	12:	 IF    bIWrappingChannelPiston2_Home AND    bIWrappingChannelPiston3_Home   THEN
		bASet4Comp:=TRUE;
		bASet3Comp:=FALSE;
		bAWrappingCone23FwdCom1:=FALSE;
		b8thConesPushed:=TRUE;
		bAFilm1Loaded_24_8Cone:=FALSE;
		bAFilm1Loaded_24_7Cone:=FALSE;
		bASensorMonitorBit3:=FALSE;
		bAConeMissErrorAtWrpConvTemp5_24:=FALSE;
		TON_8_24(IN:=FALSE);
		bWrapConvStopped4_24:=FALSE;
		TON_9_24(in:=FALSE);
		bAWrapConeCyl23_24:=FALSE;
		step4:=0;
		END_IF   sMessage_Wrapping:='Check Wrapping Piston Home  2 & 3 Reed Switch';
END_CASE


IF bAFlimNotLoaded3 AND b2_4SetHmiSelected AND bErrorReset AND bAutoModeOn THEN step4:=10; bAFlimNotLoaded3:=FALSE;HmiFilmLoadErr:=''; END_IF






IF bA6conesPushed AND CounterTilt23.CV<=3 THEN
bANextLayerStarted:=TRUE;
END_IF


IF bA3Pushed OR bA6conesPushed AND bAFirstConeAtWrapConv THEN
bAConvStartInterlock:=TRUE;
ELSE
bAConvStartInterlock:=FALSE;
END_IF

(*

IF bAConvFirstStartUnitB THEN
baConveyerStarted:=TRUE;
END_IF
IF baConveyerStarted AND



*)




IF bIWrappingCone1 AND   InterLockCounter.CV = 0  AND NOT  bQWrappingConveyorMotor THEN
 Interlockfor_1Cone_24:=TRUE;
 ELSE
 Interlockfor_1Cone_24:=FALSE; END_IF


IF bIWrappingCone1 AND   InterLockCounter.CV = 4  AND NOT  bQWrappingConveyorMotor THEN
 Interlockfor_5Cone_24:=TRUE;
 ELSE
 Interlockfor_5Cone_24:=FALSE; END_IF

IF bIWrappingCone1 AND   InterLockCounter.CV = 6  AND NOT  bQWrappingConveyorMotor THEN
 Interlockfor_7Cone_24:=TRUE;
 ELSE
 Interlockfor_7Cone_24:=FALSE; END_IF

WrappingCone1RT(CLK:=( bIWrappingCone1 AND NOT Interlockfor_1Cone_24 AND NOT Interlockfor_5Cone_24 AND NOT Interlockfor_7Cone_24 ), Q=> );

WrappingConvRT(CLK:= bQWrappingConveyorMotor , Q=> );

IF  WrappingConvRT.Q THEN
bAWrapConvStarted:=TRUE;

END_IF

IF WrappingCone1RT.Q THEN WCS1Sensed:=TRUE; END_IF

IF WCS1Sensed  (* AND bAWrapConvStarted OR bConvRunning*)  THEN
bAInterlockCountStart:=TRUE;
ELSE
bAInterlockCountStart:=FALSE;
 END_IF


IF  bQWrappingConveyorMotor AND NOT bIWrappingCone1 AND bAutoModeOn THEN
WCS1Sensed:=FALSE;
END_IF

(*TON_6(IN:=WCS1Sensed , PT:=T#0.2s , Q=> , ET=> );

IF TON_6.Q THEN bAWrapConvStarted:=FALSE; (*TON_6(in:=FALSE);*)END_IF


IF InterLockCounter.CV = 2 AND bManualModeOn THEN
TimerStartBit:=TRUE;
bAWrapConvStarted:=FALSE;
TON_10(IN:=TimerStartBit , PT:=t#0.2s , Q=> , ET=> );

 END_IF


IF TON_10.Q AND bQWrappingConveyorMotor THEN
bConvRunning:=TRUE;(*TON_10(in:=FALSE);*)
END_IF*)




IF bRowStopperIntOver THEN
bSaelUnitIntOverTemp:=TRUE;
END_IF



                                                                   (*=============== Interlock Logic for  2*4 WCS conveyor===================*)


CASE step7 OF


	0:	IF bSaelUnitIntOverTemp AND b2_4SetHmiSelected  THEN                                    (*========= need to check for reset Logic=    step7:=0    =======*)
		Step7:=Step7+1;
		END_IF

	1:	bWCSStart1_24:=TRUE;
		Step7:=Step7+1;

	2:	IF  bASealConvEnd1_24 THEN
		bSaelUnitIntOverTemp:=FALSE;
		Step7:=Step7+1;
		END_IF

	3:	bWCSStart2_24:=TRUE;
		bASealConvEnd1_24:=FALSE;
		Step7:=Step7+1;


	4:	IF bASealConvEnd2_24  THEN
		Step7:=Step7+1;
		END_IF

	5:	bWCSStart3_24:=TRUE;
		bASealConvEnd2_24:=FALSE;
		Step7:=2;

END_CASE



IF NOT bIEmergencySwitch OR bStopHmi  OR bServoOff OR bIMcStop THEN

bAWrappingConvStartAuto3_23:=FALSE;
bAWrappingConvStartAuto4_23:=FALSE;
bAWrappingConvStartAuto3:=FALSE;
bAWrappingConvStartAuto4:=FALSE;
bAWrappingConvStartAuto5:=FALSE;


		bAWrappingCone123FwdCom:=FALSE;


SealingOver1:=FALSE;

bAFilm1Loaded:=FALSE;
bAFilm2Loaded:=FALSE;
bAFilm3Loaded:=FALSE;
		WrapConvStartDly(in:=FALSE);
		bAConvRunning1:=FALSE;
		bWrapConvStopped2:=FALSE;
		TON_3(IN:=FALSE);
		TON_13_24(in:=FALSE);
		TON_4_24(IN:=FALSE);
		TON_12_24(in:=FALSE);
		bAConeMissErrorAtWrpConvTemp1_24:=FALSE;
		bAConeMissErrorAtWrpConvTemp2_24:=FALSE;
		bAWrapConeCyl123:=FALSE;

bWrapConvStopped2:=FALSE;
bWrapConvStopped3_24:=FALSE;
bWrapConvStopped4_24:=FALSE;
bWrapConvStopped4_24exp:=FALSE;


bAWrappingConvStart1_23:=FALSE;
bAWrappingConvStart4_23:=FALSE;
bAWrappingConvStart1:=FALSE;
bAWrappingConvStart2:=FALSE;
bAWrappingConvStart3:=FALSE;
bAWrappingConvStart4:=FALSE;
bAWrappingConvStart5:=FALSE;

bAconvReayTemp:=FALSE;
bAconvReayTemp2:=FALSE;
bAconvReadyTemp3:=FALSE;
bAconvReadyTemp4:=FALSE;
bAconvReadyTemp5:=FALSE;

bAWrappingConvStart1_23:=FALSE;
bACheckWrappConvError1:=FALSE;
bACheckWrappConvError2:=FALSE;
bACheckWrappConvError3:=FALSE;
bACheckWrappConvError4:=FALSE;
bACheckWrappConvError5:=FALSE;

bAWrappingConvStartAuto:=FALSE;
bAWrappingConvStartAuto2:=FALSE;
 bAWrappingConvStartAuto3:=FALSE;

bQAWrappingConveyorMotor1:=FALSE;
 bQAWrappingConveyorMotor2:=FALSE;
bQAWrappingConveyorMotor3:=FALSE;
 bQAWrappingConveyorMotor4:=FALSE;
bQAWrappingConveyorMotor5:=FALSE;

WrapConvStartDly3_23(IN:= FALSE);

bAConvRunning1:=FALSE;
 bAConvStartBit:=FALSE;

bASensorMonitorBit1:=FALSE;
bASensorMonitorBit2:=FALSE;
 bASensorMonitorBit3:=FALSE;

bASet1Comp:=FALSE;
bASet3Comp:=FALSE;
bASet2Comp:=FALSE;
bASet4Comp:=FALSE;

bAWrapConeCyl3:=FALSE;
bAWrapConeCyl123:=FALSE;
bAWrapConeCyl23_24_1:=FALSE;
bAWrapConeCyl23_24:=FALSE;

WCS1Sensed:=FALSE;
bSaelUnitIntOver:=FALSE;


bASealConvEnd1:=FALSE;
bASealConvEnd2:=FALSE;

InterLockCounter.RESET:=TRUE;
bAWrappingCone123OnAuto:=FALSE;
bAWrappingCone123_23OnAuto:=FALSE;
bQAWrappingConveyorMotor4_23:=FALSE;
bQAWrappingConveyorMotor3_23:=FALSE;


bCount_ConvLockBit2:=FALSE;
bCount_ConvLockBit:=FALSE;
bASealConvEnd1_24:=FALSE;
bASealConvEnd2_24:=FALSE;
step1:=0;
step2:=0;
step3:=0;
step4:=0;
step5:=0;
step6:=0;
step7:=0;
bAConvStartBit:=FALSE;

bA3Pushed:=FALSE;
b4thConePushed:=FALSE;
b6thConePushed_24:=FALSE;

bWCSStart1_24:=FALSE;
bWCSStart2_24:=FALSE;
bWCSStart3_24:=FALSE;

TON_6_24(IN:=FALSE) ;

TON_8_24(IN:=FALSE) ;
TON_9_24(IN:=FALSE);
TON_10_24(IN:=FALSE);



		bAWrappingCone3FwdCom:=FALSE;
		bAFilm1Loaded_24_4Cone:=FALSE;
		bASensorMonitorBit1:=FALSE;
		bWrapConvStopped4_24exp:=FALSE;
 		TON_5_24(IN:=FALSE);
		TON_11_24(in:=FALSE);
		bAWrappingCone3OnAuto:=FALSE;
		bAFilmLoadedCom:=FALSE;
		bAConeMissErrorAtWrpConvTemp3_24:=FALSE;
		bWrapConvStopped4_24exp:=FALSE;
		bAWrapConeCyl3:=FALSE;
		bA4thWrappOver:=FALSE;

bAWrappingCone23FwdCom:=FALSE;
		bAFilm1Loaded_24_6Cone:=FALSE;
		bAFilm1Loaded_24_5Cone:=FALSE;
		bASensorMonitorBit2:=FALSE;
		bAConeMissErrorAtWrpConvTemp4_24:=FALSE;
		 TON_6_24(IN:=FALSE) ;
		TON_10_24(in:=FALSE);
		bWrapConvStopped3_24:=FALSE;
		bAWrapConeCyl23_24:=FALSE;
		bAWrapConeCyl23_24_1:=FALSE;
		bA6thConeWrappOver:=FALSE;


		bAWrappingCone23FwdCom1:=FALSE;
		b8thConesPushed:=FALSE;
		bAFilm1Loaded_24_8Cone:=FALSE;
		bAFilm1Loaded_24_7Cone:=FALSE;
		bASensorMonitorBit3:=FALSE;
		bAConeMissErrorAtWrpConvTemp5_24:=FALSE;
		TON_8_24(IN:=FALSE);
		bWrapConvStopped4_24:=FALSE;
		TON_9_24(in:=FALSE);
		bAWrapConeCyl23_24:=FALSE;
		bAWrapConeCyl23_24:=FALSE;
		bA8thConeWrappOver:=FALSE;

		bSaelUnitIntOverTemp:=FALSE;

ELSE
InterLockCounter.RESET:=FALSE;
END_IF
END_PROGRAM

(* POU Auto/Sealing_Conveyor_24, ST *)
PROGRAM Sealing_Conveyor_24
VAR
	bA3ConeSealStarted: BOOL;
	bA3ConeSealComp: BOOL;

	bAConeCountSenEnable1: BOOL;
	CTU_1: CTU;
	step1: INT;
	step2: INT;
	bA4thConeSealStarted: BOOL;
	bA4thConeSealComp: BOOL;

	ConvStopDly1: TON;
	bAColoumnConeDeducted: BOOL;
	step3: INT;
	bA6thConeSealStarted: BOOL;
	bA6thConeSealComp: BOOL;

	ConvStopDly2: TON;
	ConvStopDly3: TON;
	bA8thConeSealStarted: BOOL;
	bA8thConeSealComp: BOOL;
	step4: INT;

	ConvStopDly4: TON;
	bQASealingConveyor1: BOOL;
	bQASealingConveyor2: BOOL;
	bQASealingConveyor3: BOOL;
	bQASealingConveyor4: BOOL;
	Step5: INT;
	bSealConvIntOverTemp: BOOL;
	CTU_1AlarmOnly: CTU;

	bCountLockBit_24: BOOL;
	CTU_1_24: CTU;
	CTU_1_24_AlarmOnly: CTU;
	bQASealingConveyor5: BOOL;
	bQASealingConveyor6: BOOL;
	bQASealingConveyor7: BOOL;
	bQASealingConveyor8: BOOL;
	bSecSetStarted_24: BOOL;
	SealCountBit_24: BOOL;
	bCountLock1: BOOL;
	bCountLock5_24: BOOL;
	bCountLock6_24: BOOL;
	bCountLock2_24: BOOL;
	bCountLock3_24: BOOL;
	bCountLock4_24: BOOL;
	bCountLock1_24: BOOL;
	bCountLock7_24: BOOL;
	bCountLock8_24: BOOL;
	bCountLock: BOOL;
	bAConeMissAtSealConv4_24: BOOL;
	tSealStopDly_24: TIME;
	bAConeMissAtSealConv1_24: BOOL;
	bAConeMissAtSealConv2_24: BOOL;
	bAConeMissAtSealConv3_24: BOOL;
	bQASealingConveyor9: BOOL;
	bAConeMissAtSealConv5_24: BOOL;
	Timer1: TON;
	bA4ConeCrossed_24: BOOL;
	bA6ConeCrossed_24: BOOL;
	bA8ConeCrossed_24: BOOL;
	ConvStopDly01_24: TON;
	bQASealingConveyor123_24: BOOL;
	bQASealingConveyor1234_24: BOOL;
	ConvStopDly02_24: TON;
	ConvStopDly03_24: TON;
	ConvStopDly04_24: TON;
	bQASealingConveyor123456_24: BOOL;
	bQASealingConveyor12345678_24: BOOL;
	bQASealingConveyor10: BOOL;
	bQASealingConveyor11: BOOL;
	bAConeMissAtSealConv6_24: BOOL;
	bAConeMissAtSealConv7_24: BOOL;
	bQASealingConveyor12: BOOL;
	bAConeMissAtSealConv8_24: BOOL;
	bCountLock10_24: BOOL;
	bCountLock9_24: BOOL;
	bCountLock123_24: BOOL;
	bCountLock1234_24: BOOL;
	ConvStopDly06_24: TON;
	bQASealingConveyor1234_24_1: BOOL;
	bQASealingConveyor123_24_1: BOOL;
	ConvStopDly07_24: TON;
	ConvStopDly08_24: TON;
	bQASealingConveyor123456_24_1: BOOL;
	ConvStopDly09_24: TON;
	bQASealingConveyor12345678_24_1: BOOL;
	ConvStopDly11_24: TON;
	bQASealingConveyorSample123_24: BOOL;
	bQASealingConveyorSample1234_24: BOOL;
	bQASealingConveyorSample123456_24: BOOL;
	bQASealingConveyorSample12345678_24: BOOL;
	bCountLock_24: BOOL;
	bCountLock123_24_1: BOOL;
	bCountLock1234_24_1: BOOL;
	bCountLock123456_24_1: BOOL;
	bCountLock11_24: BOOL;
	bCountLock123456_24: BOOL;
	bCountLock12345678_24_1: BOOL;
	bCountLock12_24: BOOL;
	bCountLock12345678_24: BOOL;
	bSet1Started_24: BOOL;
	bSet2Started_24: BOOL;
	bSet3Started_24: BOOL;
	bSet4Started_24: BOOL;
	bCountLockBit1_24: BOOL;
	bCountLockBit2_24: BOOL;
	bCountLockBit3_24: BOOL;
	bCountLockBit4_24: BOOL;
	bAConeMissAtSealConv01_24: BOOL;
	bACounter_24Reset: BOOL;
	bACounter_24: BOOL;
END_VAR
							(*###########################Sealing Conveyor On Bit######################### *)

bQASealingConveyorMotor1:= (bQASealingConveyor1 OR bQASealingConveyor2 OR bQASealingConveyor3 OR bQASealingConveyor4 OR bQASealingConveyor5 OR bQASealingConveyor6 OR bQASealingConveyor7 OR bQASealingConveyor8 OR bQASealingConveyor9 OR bQASealingConveyor10 OR bQASealingConveyor11 OR bQASealingConveyor12 );

							(*###########################Sealing Conveyor Count interlock t######################### *)

IF bQASealingConveyorMotor AND bSet1Started_24  AND CTU_1_24_AlarmOnly.CV=3 THEN bCountLockBit1_24:=TRUE; END_IF
IF bQASealingConveyorMotor AND bSet2Started_24  AND CTU_1_24_AlarmOnly.CV=4 THEN bCountLockBit2_24:=TRUE; END_IF
IF bQASealingConveyorMotor AND bSet3Started_24  AND CTU_1_24_AlarmOnly.CV=6 THEN bCountLockBit3_24:=TRUE; END_IF
IF bQASealingConveyorMotor AND bSet4Started_24  AND CTU_1_24_AlarmOnly.CV=8 THEN bCountLockBit4_24:=TRUE; END_IF


IF bQASealingConveyorMotor AND bIConeCountSensor AND b2_4SetHmiSelected  AND NOT bCountLockBit1_24 AND NOT bCountLockBit2_24
 AND NOT bCountLockBit3_24 AND NOT bCountLockBit4_24  THEN
	bAConeCountSenEnable1:=TRUE;
ELSE
	bAConeCountSenEnable1:=FALSE;
END_IF

CTU_1(
	CU:=bAConeCountSenEnable1 ,
	RESET:= ,
	PV:=8 ,
	Q=> ,
	CV=> );


CTU_1_24_AlarmOnly(
	CU:=(bAConeCountSenEnable1 AND NOT bCountLock_24) ,
	RESET:=bACounter_24Reset OR bACounter_24 ,
	PV:=8 ,
	Q=> ,
	CV=> );


IF bQASealingConveyorMotor AND bSecSetStarted_24 AND  CTU_1.CV=8 THEN SealCountBit_24:=TRUE; END_IF


				(*############################  1,2,3rd  Cone Sealing Conveyor   ############################*)


CASE step1 OF

		0:	IF bAutoModeOn AND b2_4SetHmiSelected AND  bA3ConeWrappOver_24 AND bQASealingSeparatorYAxisPistonValve THEN
			bA3ConeSealStarted:=TRUE;
			CTU_1.RESET:=TRUE;
			bACounter_24:=TRUE;
			 tSealStopDly_24:=t#2.5s;
			ConvStopDly1(IN:=FALSE); ConvStopDly06_24(in:=FALSE);
			 step1:=step1+1; END_IF

		1:	IF NOT bAPauseSeq THEN step1:=step1+1; END_IF

		2:	IF bAutoModeOn AND b2_4SetHmiSelected AND  bA3ConeSealStarted AND bISealingSeparatorXAxisEnd THEN
			bA3ConeSealComp:=TRUE;
			bAConeAtMatrixEr_01:=TRUE;
			CTU_1.RESET:=FALSE;
			bACounter_24:=FALSE;
		 	Timer1(IN:=FALSE);
			step1:=step1+1; END_IF

		3:	IF NOT bAPauseSeq THEN step1:=step1+1; END_IF

		4:	IF bAutoModeOn AND   bA3ConeSealComp AND (bSealConvStart1_24 OR bSealConvStart3_24)  AND NOT bASealSepaX_axisRsError THEN
			bQASealingConveyor1:=TRUE;
			ConvStopDly1(in:=FALSE);
			ConvStopDly06_24(in:=FALSE);
			bSet1Started_24:=TRUE;
			 step1:=step1+1; END_IF

		5:	ConvStopDly1(in:=FALSE);
			 step1:=step1+1;

		6:	IF NOT bAPauseSeq THEN  step1:=step1+1; END_IF

		7:	IF CTU_1_24_AlarmOnly.CV>=3 THEN
			bSealConvStart1_24:=FALSE;
			bSealConvStart3_24:=FALSE;
			bA3ConeCrossed_24:=TRUE;
			bA3ConeSealComp:=FALSE;
			bA3ConeSealStarted:=FALSE;
			 step1:=step1+1; END_IF

		8:	(*IF bIColumnconeDetection THEN*)
		step1:=step1+1;
		(*END_IF*)

		9:	ConvStopDly1(IN:=TRUE , PT:= t#0.5s , Q=> , ET=> );
			IF ConvStopDly1.Q THEN step1:=step1+1; END_IF

		10:	 step1:=step1+1;

		11:	bQASealingConveyor1:=FALSE;
			bQASealingConveyor5:=FALSE;
			bQASealingConveyor6:=FALSE;
			bA3ConeSealComp:=FALSE;
			bA3ConeSealStarted:=FALSE;
			bCountLock1_24:=FALSE;
			bCountLock5_24:=FALSE;
			bCountLock6_24:=FALSE;
			bA3ConeCrossed_24:=FALSE;
			bQASealingConveyor123_24:=FALSE;
			bAConeMissAtSealConv2_24:=FALSE;
			ConvStopDly01_24(in:=FALSE);
			bQASealingConveyorSample123_24:=FALSE;
			bQASealingConveyor123_24_1:=FALSE;
			bSet1Started_24:=FALSE;
			bCountLockBit1_24:=FALSE;
			bCountLock123_24:=FALSE;
			bCountLock123_24_1:=FALSE;
			ConvStopDly06_24(in:=FALSE);
			bAConeAtMatrixEr_01:=FALSE;
			step1:=step1+1;


		12:	IF NOT bAPauseSeq THEN step1:=step1+1; END_IF

		13:	step1:=0;

END_CASE

				(*############################  4th Cone Sealing Conveyor   #####################*)

CASE step2 OF

	0:	IF bAutoModeOn AND b2_4SetHmiSelected AND  bA4thWrappOver AND bQASealingSeparatorYAxisPistonValve THEN
		bA4thConeSealStarted:=TRUE;
		 tSealStopDly_24:=t#2.5s;
		ConvStopDly2(IN:=FALSE);
		bQASealingConveyor123_24_1:=FALSE;
		ConvStopDly06_24(in:=FALSE);
		step2:=step2+1;
		END_IF

	1:	IF NOT bAPauseSeq THEN step2:=step2+1; END_IF

	2:	IF bAutoModeOn AND b2_4SetHmiSelected AND  bA4thConeSealStarted AND bISealingSeparatorXAxisEnd THEN
		bA4thConeSealComp:=TRUE;
		bAConeAtMatrixEr_02:=TRUE;
		step2:=step2+1;
		END_IF

	3:	IF NOT bAPauseSeq THEN step2:=step2+1; END_IF

	4:	IF bAutoModeOn AND   bA4thConeSealComp  AND NOT bAPauseSeq AND NOT bASealSepaX_axisRsError THEN
		bQASealingConveyor2:=TRUE;
		bSet2Started_24:=TRUE;
		step2:=step2+1;
		END_IF

	5:	ConvStopDly2(in:=FALSE);
		ConvStopDly07_24(in:=FALSE);
		step2:=step2+1;

	6:	IF NOT bAPauseSeq THEN step2:=step2+1; END_IF

	7:	IF CTU_1_24_AlarmOnly.CV>=4 THEN
		bA4thConeSealComp:=FALSE;
		bA4thConeSealStarted:=FALSE;
		bA4ConeCrossed_24:=TRUE;
		step2:=step2+1;
		END_IF

	8:	(*IF NOT bAPauseSeq THEN step2:=step2+1; END_IF*) step2:=step2+1;

	9:	IF bIColumnconeDetection THEN
		ConvStopDly2(IN:=TRUE , PT:=t#2s , Q=> , ET=> );
		IF ConvStopDly2.Q THEN    step2:=step2+1; END_IF
		END_IF

	10:	 step2:=step2+1;

	11:	bQASealingConveyor2:=FALSE;
		bQASealingConveyor9:=FALSE;
		bAColumnPushPistonStart1:=TRUE;
		bASealConvEnd1_24:=TRUE;
		bA4ConeCrossed_24:=FALSE;
		bQASealingConveyor1234_24:=FALSE;
		bAConeMissAtSealConv3_24:=FALSE;
		bAConeMissAtSealConv4_24:=FALSE;
		bQASealingConveyor10:=FALSE;
		ConvStopDly02_24(in:=FALSE);
		bQASealingConveyor9:=FALSE;
		ConvStopDly07_24(in:=FALSE);
		bQASealingConveyorSample1234_24:=FALSE;
		bQASealingConveyor1234_24_1:=FALSE;
		bSet2Started_24:=FALSE;
		bCountLockBit2_24:=FALSE;
		bCountLock1234_24_1:=FALSE;
		bCountLock1234_24:=FALSE;
		bCountLock2_24:=FALSE;
		bCountLock9_24:=FALSE;
		bCountLock10_24:=FALSE;
		bAConeAtMatrixEr_02:=FALSE;
		step2:=0;


END_CASE


				(*############################  5,6th Cone Sealing Conveyor   #########################*)


CASE step3 OF

	0:	IF bAutoModeOn AND b2_4SetHmiSelected AND  bA6thConeWrappOver AND bQASealingSeparatorYAxisPistonValve THEN
		bA6thConeSealStarted:=TRUE;
		 tSealStopDly_24:=t#2.5s;
		ConvStopDly3(IN:=FALSE );
		bQASealingConveyor1234_24_1:=FALSE;
		ConvStopDly07_24(in:=FALSE);
		step3:=step3+1;
		END_IF

	1:	IF NOT bAPauseSeq THEN step3:=step3+1; END_IF

	2:	IF bAutoModeOn AND b2_4SetHmiSelected AND  bA6thConeSealStarted AND bISealingSeparatorXAxisEnd THEN
		bA6thConeSealComp:=TRUE;
		bAConeAtMatrixEr_03:=TRUE;
		step3:=step3+1;
		END_IF

	3:	IF NOT bAPauseSeq THEN step3:=step3+1; END_IF

	4:	IF bAutoModeOn AND   bA6thConeSealComp AND bSealConvStart2_24 AND NOT bAPauseSeq AND NOT bASealSepaX_axisRsError   THEN
		bQASealingConveyor3:=TRUE;
		bSet3Started_24:=TRUE;
		step3:=step3+1;
		END_IF


	5:	ConvStopDly3(in:=FALSE);
		ConvStopDly08_24(in:=FALSE);
 		step3:=step3+1;


	6:	IF NOT bAPauseSeq THEN step3:=step3+1; END_IF

	7:	IF CTU_1_24_AlarmOnly.CV>=6 THEN
		bSealConvStart2_24:=FALSE;
		bA6ConeCrossed_24:=TRUE;
		ConvStopDly3(IN:=TRUE , PT:=t#0.5s , Q=> , ET=> );
		IF ConvStopDly3.Q THEN  step3:=step3+1; END_IF
		END_IF

	8:	 step3:=step3+1;

	9:	bA6thConeSealComp:=FALSE;
		bA6thConeSealStarted:=FALSE;
		bQASealingConveyor3:=FALSE;
		bQASealingConveyor7:=FALSE;
		bA6ConeCrossed_24:=FALSE;
		bQASealingConveyor123456_24:=FALSE;
		bAConeMissAtSealConv4_24:=FALSE;
		ConvStopDly03_24(in:=FALSE);
		bAConeMissAtSealConv6_24:=FALSE;
		bQASealingConveyor11:=FALSE;
		ConvStopDly08_24(in:=FALSE);
		bQASealingConveyorSample123456_24:=FALSE;
		bSet3Started_24:=FALSE;
		bCountLockBit3_24:=FALSE;
		bCountLock3_24:=FALSE;
		bCountLock7_24:=FALSE;
		bCountLock11_24:=FALSE;
		bCountLock123456_24:=FALSE;
		bCountLock123456_24_1:=FALSE;
		bQASealingConveyor123456_24_1:=FALSE;
		bAConeAtMatrixEr_03:=FALSE;
		step3:=step3+1;

	10:	IF NOT bAPauseSeq THEN step3:=step3+1; END_IF

	11:	step3:=0;

END_CASE


				(*############################  7, 8th Cone Sealing Conveyor   #########################*)


CASE step4 OF

	0:	IF bAutoModeOn AND b2_4SetHmiSelected AND  bA8thConeWrappOver AND bQASealingSeparatorYAxisPistonValve THEN
		bA8thConeSealStarted:=TRUE;
		 tSealStopDly_24:=t#2.5s;
		ConvStopDly4(IN:=FALSE);
		step4:=step4+1;
		END_IF

	1:	IF NOT bAPauseSeq THEN step4:=step4+1; END_IF

	2:	IF bAutoModeOn AND b2_4SetHmiSelected AND  bA8thConeSealStarted AND bISealingSeparatorXAxisEnd THEN
		bA8thConeSealComp:=TRUE;
		bAConeAtMatrixEr_04:=TRUE;
		step4:=step4+1;
		END_IF

	3:	IF NOT bAPauseSeq THEN step4:=step4+1; END_IF

	4:	IF bAutoModeOn AND   bA8thConeSealComp AND NOT bAPauseSeq  AND NOT bASealSepaX_axisRsError  THEN
		bQASealingConveyor4:=TRUE;
		bSet4Started_24:=TRUE;
		step4:=step4+1;
		END_IF

	5:	ConvStopDly4(in:=FALSE);
		ConvStopDly11_24(in:=FALSE);
 		step4:=step4+1;

	6:	IF NOT bAPauseSeq THEN step4:=step4+1; END_IF

	7:	IF CTU_1_24_AlarmOnly.CV=8 THEN
		bA8thConeSealComp:=FALSE;
		bA8thConeSealStarted:=FALSE;
		bA8ConeCrossed_24:=TRUE;
		step4:=step4+1;
		END_IF

	8:	(*IF NOT bAPauseSeq THEN step4:=step4+1; END_IF*) step4:=step4+1;

	9:	IF bIColumnconeDetection THEN
		ConvStopDly4(IN:=TRUE , PT:=tSealStopDly_24 , Q=> , ET=> );
		IF ConvStopDly4.Q THEN  bACounter_24:=TRUE;   step4:=step4+1; END_IF
		END_IF

	10:	 step4:=step4+1;

	11:	bQASealingConveyor4:=FALSE;
		bQASealingConveyor8:=FALSE;
		bAColumnPushPistonStart2:=TRUE;
		bASealConvEnd2_24:=TRUE;
		CTU_1.RESET:=FALSE;
		SealCountBit_24:=FALSE;
		bA8ConeCrossed_24:=FALSE;
		bQASealingConveyor12345678_24:=FALSE;
		ConvStopDly04_24(in:=FALSE);
		bAConeMissAtSealConv7_24:=FALSE;
		bQASealingConveyor12:=FALSE;
		bAConeMissAtSealConv8_24:=FALSE;
		ConvStopDly11_24(in:=FALSE);
		bQASealingConveyor12345678_24_1:=FALSE;
		bQASealingConveyorSample12345678_24:=FALSE;
		bSet4Started_24:=FALSE;
		bCountLockBit4_24:=FALSE;
		bCountLock4_24:=FALSE;
		bCountLock8_24:=FALSE;
		bCountLock12_24:=FALSE;
		bCountLock12345678_24:=FALSE;
		bCountLock12345678_24_1:=FALSE;
		bAConeAtMatrixEr_04:=FALSE;
		step4:=0;
		bACounter_24:=FALSE;
END_CASE




IF bRowStopperIntOver  AND b2_4SetHmiSelected THEN
bSealConvIntOverTemp:=TRUE;
END_IF


CASE step5 OF


0:	IF bSealConvIntOverTemp  AND b2_4SetHmiSelected THEN
	Step5:=Step5+1;
	END_IF

1:	IF NOT bIColumnconeDetection THEN
	bSealConvStart1_24:=TRUE;
	Step5:=Step5+1;
	END_IF

2:	IF  CTU_1_24_AlarmOnly.CV=4 THEN

	Step5:=Step5+1;
	END_IF

3:	IF bIColumnconeDetection THEN
	Step5:=Step5+1;
	END_IF

4:	IF bAFirstSetToMatrix  THEN
	bSealConvStart2_24:=TRUE;
	Step5:=Step5+1;
	END_IF

5:	IF	CTU_1_24_AlarmOnly.CV=8 THEN
	bAFirstSetToMatrix:=FALSE;
	Step5:=Step5+1;
	END_IF

6:	IF bIColumnconeDetection THEN
	Step5:=Step5+1;
	END_IF

7:	IF bASecondSetToMatrix THEN
	bSealConvStart3_24:=TRUE;
	Step5:=Step5+1;
	END_IF

8:	bASecondSetToMatrix:=FALSE;
	Step5:=1;
END_CASE


(*

	IF bAresetHmi THEN
	Step5:=0;
	bSealConvStart1_24:=FALSE;
	bSealConvStart2_24:=FALSE;
	bASecondSetToMatrix:=FALSE;
	bAFirstSetToMatrix:=FALSE;
	bSealConvStart3_24:=FALSE;
	END_IF
*)

									(*--------------------------------------------------------Alarm Sequence---------------------------------------------------------*)

IF bQASealingConveyor1 AND CTU_1_24_AlarmOnly.CV =3  THEN  bCountLock1_24:=TRUE; END_IF
IF bQASealingConveyor5 AND CTU_1_24_AlarmOnly.CV =3  THEN  bCountLock5_24:=TRUE; END_IF
IF bQASealingConveyor6 AND CTU_1_24_AlarmOnly.CV =3  THEN  bCountLock6_24:=TRUE; END_IF
IF bQASealingConveyor123_24	   AND CTU_1_24_AlarmOnly.CV=3 THEN  bCountLock123_24:=TRUE; END_IF
IF bQASealingConveyor123_24_1 AND CTU_1_24_AlarmOnly.CV=3 THEN bCountLock123_24_1:=TRUE;END_IF


IF bQASealingConveyor2 AND CTU_1_24_AlarmOnly.CV =4  THEN  bCountLock2_24:=TRUE; END_IF
IF bQASealingConveyor10 AND CTU_1_24_AlarmOnly.CV =4  THEN  bCountLock10_24:=TRUE; END_IF
IF bQASealingConveyor1234_24_1 AND CTU_1_24_AlarmOnly.CV =4 THEN bCountLock1234_24_1:=TRUE; END_IF
IF bQASealingConveyor9 AND CTU_1_24_AlarmOnly.CV =4  THEN  bCountLock9_24:=TRUE; END_IF
IF bQASealingConveyor1234_24 AND CTU_1_24_AlarmOnly.CV =4  THEN  bCountLock1234_24:=TRUE; END_IF


IF bQASealingConveyor3 AND CTU_1_24_AlarmOnly.CV =6  THEN  bCountLock3_24:=TRUE; END_IF
IF bQASealingConveyor7 AND CTU_1_24_AlarmOnly.CV =6  THEN  bCountLock7_24:=TRUE; END_IF
IF bQASealingConveyor123456_24_1 AND CTU_1_24_AlarmOnly.CV =6  THEN  bCountLock123456_24_1:=TRUE; END_IF
IF bQASealingConveyor11 AND CTU_1_24_AlarmOnly.CV =6  THEN  bCountLock11_24:=TRUE; END_IF
IF bQASealingConveyor123456_24 AND CTU_1_24_AlarmOnly.CV =6  THEN  bCountLock123456_24:=TRUE; END_IF

IF bQASealingConveyor4 AND CTU_1_24_AlarmOnly.CV =8  THEN  bCountLock4_24:=TRUE; END_IF
IF bQASealingConveyor12345678_24_1 AND CTU_1_24_AlarmOnly.CV =8  THEN  bCountLock12345678_24_1:=TRUE; END_IF
IF bQASealingConveyor12 AND CTU_1_24_AlarmOnly.CV =8  THEN  bCountLock12_24:=TRUE; END_IF
IF bQASealingConveyor12345678_24 AND CTU_1_24_AlarmOnly.CV =8  THEN  bCountLock12345678_24:=TRUE; END_IF
IF bQASealingConveyor8 AND CTU_1_24_AlarmOnly.CV =8  THEN  bCountLock8_24:=TRUE; END_IF

 IF bCountLock1_24 OR bCountLock2_24 OR  bCountLock3_24 OR bCountLock4_24 OR  bCountLock5_24 OR bCountLock6_24
OR bCountLock7_24 OR bCountLock8_24 OR bCountLock9_24 OR bCountLock10_24 OR bCountLock11_24 OR bCountLock12_24
OR bCountLock123_24 OR  bCountLock1234_24  OR  bCountLock123456_24 OR  bCountLock12345678_24
OR bCountLock123_24_1 OR bCountLock1234_24_1 OR bCountLock123456_24_1 OR bCountLock12345678_24_1
THEN
 bCountLock_24:=TRUE;
 ELSE
bCountLock_24:=FALSE;
 END_IF

						(*--------------------------------------------------------Alarm Sequence Cone 2 Missing---------------------------------------------------------*)


IF bQASealingConveyor1 AND NOT bIConeCountSensor AND  NOT bAPauseSeq  THEN ConvStopDly06_24(IN:=TRUE , PT:=t#6s , Q=> , ET=> );END_IF
IF ConvStopDly06_24.Q THEN bQASealingConveyor123_24_1:=TRUE; bQASealingConveyor1:=FALSE; END_IF

IF bQASealingConveyor123_24_1    AND  (CTU_1_24_AlarmOnly.CV ) <3  AND  NOT bAPauseSeq THEN
bAConeMissAtSealConv01_24:=TRUE;
bQASealingConveyor1:=FALSE;
bQASealingConveyor123_24_1:=FALSE;
ConvStopDly06_24(in:=FALSE);
SealConeMiss:=' Cone  Missing From Sealing Conveyor';
END_IF
IF bAConeMissAtSealConv01_24 AND bErrorReset THEN
bQASealingConveyor5:=TRUE;
bAConeMissAtSealConv01_24:=FALSE;
Step1:=5;  (*tSealStopDly_24:=t#4s;*)
SealConeMiss:='Continue Machine Operation'; END_IF



						(*--------------------------------------------------------Alarm Sequence Cone 3 Missing---------------------------------------------------------*)



IF bQASealingConveyor5 OR bQASealingConveyor123_24    AND  (CTU_1_24_AlarmOnly.CV ) <3  AND  NOT bAPauseSeq  THEN
bAConeMissAtSealConv2_24:=TRUE;
bQASealingConveyor5:=FALSE;
bQASealingConveyor6:=FALSE;
bQASealingConveyor123_24:=FALSE;
ConvStopDly01_24(in:=FALSE);
bQASealingConveyorSample123_24:=FALSE;
SealConeMiss:=' Cone  Missing From Sealing Conveyor';
 END_IF
IF bAConeMissAtSealConv2_24 AND bErrorReset THEN
bQASealingConveyor6:=TRUE;  Step1:=5;  tSealStopDly_24:=t#4s;
SealConeMiss:='Continue Machine Operation'; bAConeMissAtSealConv2_24:=FALSE; END_IF

IF bQASealingConveyor6 THEN ConvStopDly01_24(IN:=TRUE , PT:=t#6s , Q=> , ET=> ); bQASealingConveyorSample123_24:=TRUE; END_IF
IF ConvStopDly01_24.Q THEN bQASealingConveyor123_24:=TRUE; END_IF



					(*--------------------------------------------------------Alarm Sequence Cone 4 Missing---------------------------------------------------------*)



IF bQASealingConveyor2 AND NOT bIConeCountSensor  AND  NOT bAPauseSeq THEN ConvStopDly07_24(IN:=TRUE , PT:=t#5s , Q=> , ET=> ); END_IF
IF ConvStopDly07_24.Q THEN bQASealingConveyor1234_24_1:=TRUE; bQASealingConveyor2:=FALSE; END_IF

IF bQASealingConveyor1234_24_1  AND  bIColumnconeDetection  AND  (CTU_1_24_AlarmOnly.CV ) <4  AND(CTU_1_24_AlarmOnly.CV ) =3 AND  NOT bAPauseSeq THEN
bAConeMissAtSealConv3_24:=TRUE;
bQASealingConveyor2:=FALSE;
bQASealingConveyor1234_24_1:=FALSE;
ConvStopDly07_24(in:=FALSE);
SealConeMiss:=' Cone  Missing From Sealing Conveyor';
END_IF
IF bAConeMissAtSealConv3_24 AND bErrorReset THEN
bQASealingConveyor10:=TRUE;
bAConeMissAtSealConv3_24:=FALSE;
Step2:=5;  tSealStopDly_24:=t#4s;
SealConeMiss:='Continue Machine Operation'; END_IF


IF bQASealingConveyor10 OR bQASealingConveyor1234_24 AND  bIColumnconeDetection  AND  (CTU_1_24_AlarmOnly.CV ) <4 AND (CTU_1_24_AlarmOnly.CV ) =3 AND  NOT bAPauseSeq   THEN
bAConeMissAtSealConv4_24:=TRUE;
bQASealingConveyor10:=FALSE;
bQASealingConveyor1234_24:=FALSE;
ConvStopDly02_24(in:=FALSE);
bQASealingConveyor9:=FALSE;
bQASealingConveyorSample1234_24:=FALSE;
SealConeMiss:=' Cone  Missing From Sealing Conveyor';
 END_IF
IF bAConeMissAtSealConv4_24 AND bErrorReset THEN
bQASealingConveyor9:=TRUE;  Step2:=5;  tSealStopDly_24:=t#4s;
SealConeMiss:='Continue Machine Operation'; bAConeMissAtSealConv4_24:=FALSE; END_IF

IF bQASealingConveyor9 THEN ConvStopDly02_24(IN:=TRUE , PT:=t#6s , Q=> , ET=> ); bQASealingConveyorSample1234_24:=TRUE;END_IF
IF ConvStopDly02_24.Q THEN bQASealingConveyor1234_24:=TRUE; END_IF



					(*--------------------------------------------------------Alarm Sequence Cone 6 Missing---------------------------------------------------------*)


IF bQASealingConveyor3 AND NOT bIConeCountSensor  AND  NOT bAPauseSeq THEN ConvStopDly08_24(IN:=TRUE , PT:=t#5s , Q=> , ET=> ); END_IF
IF ConvStopDly08_24.Q THEN bQASealingConveyor123456_24_1:=TRUE; bQASealingConveyor3:=FALSE; END_IF

IF bQASealingConveyor123456_24_1    AND  (CTU_1_24_AlarmOnly.CV ) <6  AND  (CTU_1_24_AlarmOnly.CV ) >=4  AND  NOT bAPauseSeq THEN
bAConeMissAtSealConv5_24:=TRUE;
bQASealingConveyor3:=FALSE;
ConvStopDly08_24(in:=FALSE);
bQASealingConveyor123456_24_1:=FALSE;
SealConeMiss:=' Cone  Missing From Sealing Conveyor';
END_IF
IF bAConeMissAtSealConv5_24 AND bErrorReset THEN
bQASealingConveyor11:=TRUE;
bAConeMissAtSealConv5_24:=FALSE;
Step3:=5;  tSealStopDly_24:=t#4s;
SealConeMiss:='Continue Machine Operation';
END_IF

IF bQASealingConveyor11  OR bQASealingConveyor123456_24   AND  (CTU_1_24_AlarmOnly.CV ) <6 AND  (CTU_1_24_AlarmOnly.CV ) >=4 AND  NOT bAPauseSeq   THEN
bAConeMissAtSealConv6_24:=TRUE;
bQASealingConveyor11:=FALSE;
bQASealingConveyor123456_24:=FALSE;
ConvStopDly03_24(in:=FALSE);
bQASealingConveyor7:=FALSE;
bQASealingConveyorSample123456_24:=FALSE;
SealConeMiss:=' Cone  Missing From Sealing Conveyor';
 END_IF
IF bAConeMissAtSealConv6_24 AND bErrorReset THEN
bQASealingConveyor7:=TRUE;  Step3:=5;  tSealStopDly_24:=t#4s;
SealConeMiss:='Continue Machine Operation'; bAConeMissAtSealConv6_24:=FALSE; END_IF

IF bQASealingConveyor7 THEN ConvStopDly03_24(IN:=TRUE , PT:=t#6s , Q=> , ET=> ); bQASealingConveyorSample123456_24:=TRUE;END_IF
IF ConvStopDly03_24.Q THEN bQASealingConveyor123456_24:=TRUE; END_IF


		                            (*--------------------------------------------------------Alarm Sequence Cone 8 Missing---------------------------------------------------------*)


IF bQASealingConveyor4 AND NOT bIConeCountSensor  AND  NOT bAPauseSeq THEN ConvStopDly11_24(IN:=TRUE , PT:=t#5s , Q=> , ET=> ); END_IF
IF ConvStopDly11_24.Q THEN bQASealingConveyor12345678_24_1:=TRUE; bQASealingConveyor4:=FALSE; END_IF


IF bQASealingConveyor12345678_24_1  AND  bIColumnconeDetection  AND  (CTU_1_24_AlarmOnly.CV ) <8 AND  (CTU_1_24_AlarmOnly.CV ) >=6  AND  NOT bAPauseSeq THEN
bAConeMissAtSealConv7_24:=TRUE;
bQASealingConveyor4:=FALSE;
ConvStopDly11_24(in:=FALSE);
bQASealingConveyor12345678_24_1:=FALSE;
SealConeMiss:=' Cone  Missing From Sealing Conveyor';
END_IF
IF bAConeMissAtSealConv7_24 AND bErrorReset THEN
bQASealingConveyor12:=TRUE;
bAConeMissAtSealConv7_24:=FALSE;
Step4:=5;  tSealStopDly_24:=t#4s;
SealConeMiss:='Continue Machine Operation'; END_IF


IF bQASealingConveyor12 OR bQASealingConveyor12345678_24  AND  bIColumnconeDetection  AND  (CTU_1_24_AlarmOnly.CV ) <8 AND  (CTU_1_24_AlarmOnly.CV ) >=6
AND  NOT bAPauseSeq THEN
bAConeMissAtSealConv8_24:=TRUE;
bQASealingConveyor12:=FALSE;
bQASealingConveyor12345678_24:=FALSE;
ConvStopDly04_24(in:=FALSE);
bQASealingConveyor8:=FALSE;
bQASealingConveyorSample12345678_24:=FALSE;
SealConeMiss:=' Cone  Missing From Sealing Conveyor';
 END_IF
IF bAConeMissAtSealConv8_24 AND bErrorReset THEN
bQASealingConveyor8:=TRUE;  Step4:=5;  tSealStopDly_24:=t#4s;
SealConeMiss:='Continue Machine Operation'; bAConeMissAtSealConv8_24:=FALSE; END_IF

IF bQASealingConveyor8 THEN ConvStopDly04_24(IN:=TRUE , PT:=t#6s , Q=> , ET=> ); bQASealingConveyorSample12345678_24:=TRUE; END_IF
IF ConvStopDly04_24.Q THEN bQASealingConveyor12345678_24:=TRUE; END_IF



									(*##############################Alarm Sequence in HMI#################################*)


IF bAConeMissAtSealConv01_24 OR bAConeMissAtSealConv2_24 OR bAConeMissAtSealConv3_24 OR bAConeMissAtSealConv8_24
OR bAConeMissAtSealConv4_24 OR bAConeMissAtSealConv5_24 OR bAConeMissAtSealConv6_24 OR bAConeMissAtSealConv7_24  THEN
 bQSealBitAlert:=TRUE; END_IF

IF bQSealBitAlert   AND bErrorReset   THEN   bQSealBitAlert:=FALSE; END_IF

IF bQASealingConveyor123_24_1 OR  bQASealingConveyor123_24 OR bQASealingConveyor1234_24_1 OR bQASealingConveyor123456_24_1
OR bQASealingConveyor12345678_24 OR bQASealingConveyorSample12345678_24 OR bQASealingConveyorSample123456_24 OR
 bQASealingConveyorSample1234_24 OR bQASealingConveyorSample123_24 THEN
  bQSealBitAlert_24:=TRUE; ELSE  bQSealBitAlert_24:=FALSE;  END_IF

IF bQASealingConveyor1 OR bQASealingConveyor2 OR bQASealingConveyor3 OR bQASealingConveyor4 OR bQASealingConveyor5 OR
bQASealingConveyor6 OR bQASealingConveyor7 OR bQASealingConveyor8 OR bQASealingConveyor9 OR bQASealingConveyor10 OR
bQASealingConveyor11 OR bQASealingConveyor12   THEN SealConeMissAlet_24:= TRUE; ELSE SealConeMissAlet_24:= FALSE; END_IF



IF NOT bIEmergencySwitch OR bStopHmi  OR bServoOff OR bIMcStop THEN
bQSealBitAlert:=FALSE;
bQSealBitAlert_24:=FALSE;
bACounter_24Reset:=TRUE;
CTU_1.RESET:=TRUE;

bAConeMissAtSealConv01_24:=FALSE;
bAConeMissAtSealConv2_24 :=FALSE;
bAConeMissAtSealConv3_24:=FALSE;
bAConeMissAtSealConv4_24:=FALSE;
bAConeMissAtSealConv5_24:=FALSE;
bAConeMissAtSealConv6_24:=FALSE;
bAConeMissAtSealConv7_24:=FALSE;
bAConeMissAtSealConv8_24:=FALSE;

bQASealingConveyor1:=FALSE;
bQASealingConveyor2:=FALSE;
bQASealingConveyor3:=FALSE;
bQASealingConveyor4:=FALSE;
bQASealingConveyor5:=FALSE;
bQASealingConveyor6:=FALSE;
bQASealingConveyor7:=FALSE;
bQASealingConveyor8:=FALSE;
bQASealingConveyor9:=FALSE;
bQASealingConveyor10:=FALSE;
bQASealingConveyor11:=FALSE;
bQASealingConveyor12:=FALSE;

bQASealingConveyor123_24:=FALSE;
bQASealingConveyor1234_24:=FALSE;
bQASealingConveyor123456_24:=FALSE;
bQASealingConveyor12345678_24:=FALSE;

bQASealingConveyor123_24_1:=FALSE;
 bQASealingConveyor1234_24_1:=FALSE;
 bQASealingConveyor123456_24_1:=FALSE;
 bQASealingConveyor12345678_24_1:=FALSE;

bQASealingConveyorSample123_24 :=FALSE;
bQASealingConveyorSample1234_24 :=FALSE;
bQASealingConveyorSample123456_24 :=FALSE;
bQASealingConveyorSample12345678_24:=FALSE;

bCountLock1_24:=FALSE;
bCountLock2_24:=FALSE;
bCountLock3_24:=FALSE;
bCountLock4_24:=FALSE;
bCountLock5_24:=FALSE;
bCountLock6_24:=FALSE;
bCountLock7_24:=FALSE;
bCountLock8_24:=FALSE;
bCountLock9_24:=FALSE;
bCountLock10_24:=FALSE;
bCountLock11_24:=FALSE;
bCountLock12_24:=FALSE;

bCountLock123_24:=FALSE;
bCountLock1234_24:=FALSE;
bCountLock123456_24:=FALSE;
bCountLock12345678_24:=FALSE;

bCountLock123_24_1:=FALSE;
bCountLock1234_24_1:=FALSE;
bCountLock123456_24_1:=FALSE;
bCountLock12345678_24_1:=FALSE;

bCountLockBit1_24:=FALSE;
bCountLockBit2_24:=FALSE;
bCountLockBit3_24:=FALSE;
bCountLockBit4_24:=FALSE;

Step1:=0;
Step2:=0;
Step3:=0;
Step4:=0;
Step5:=0;

bCountLock_24:=FALSE;

ConvStopDly1(IN:=FALSE);
ConvStopDly2(IN:=FALSE);
ConvStopDly3(IN:=FALSE);
ConvStopDly4(IN:=FALSE);

ConvStopDly01_24(in:=FALSE);
ConvStopDly02_24(in:=FALSE);
ConvStopDly03_24(in:=FALSE);
ConvStopDly04_24(in:=FALSE);
ConvStopDly06_24(in:=FALSE);
ConvStopDly07_24(in:=FALSE);
ConvStopDly08_24(in:=FALSE);
ConvStopDly09_24(in:=FALSE);
ConvStopDly11_24(in:=FALSE);

bSet1Started_24:=FALSE;
bSet2Started_24:=FALSE;
bSet3Started_24:=FALSE;
bSet4Started_24:=FALSE;

bSealConvStart1_24:=FALSE;
bSealConvStart2_24:=FALSE;
bSealConvStart3_24:=FALSE;


bA3ConeCrossed_24:=FALSE;
bA4ConeCrossed_24:=FALSE;
bA6ConeCrossed_24:=FALSE;
bA8ConeCrossed_24:=FALSE;


bA3ConeSealComp:=FALSE;
bA4thConeSealComp:=FALSE;
bA6thConeSealComp:=FALSE;
bA8thConeSealComp:=FALSE;

bA3ConeSealStarted:=FALSE;
bA4thConeSealStarted:=FALSE;
bA6thConeSealStarted:=FALSE;
bA8thConeSealStarted:=FALSE;

bAConeAtMatrixEr_01:=FALSE;
		bAConeAtMatrixEr_02:=FALSE;
		bAConeAtMatrixEr_03:=FALSE;
		bAConeAtMatrixEr_04:=FALSE;

bSealConvIntOverTemp:=FALSE;

ELSE
bACounter_24Reset:=FALSE;
CTU_1.RESET:=FALSE;
END_IF
END_PROGRAM

(* POU ERROR_1, ST *)
PROGRAM ERROR_1
VAR
	bfAlarmbit1: BOOL;
	sAlarmBuffer: ARRAY[1..5] OF STRING;
	sAlarmArray: ARRAY[0..50] OF STRING;
	ifAlarmStep: INT;
	k: INT;
	sAlarmValue: STRING;
	bfAlarmGenerated: BOOL;
	sAlarm1: STRING(80);
	bfAlarmbit2: BOOL;
	bfAlarmbit3: BOOL;
	bfAlarmbit4: BOOL;
	bfAlarmbit5: BOOL;
	sAlarm2: STRING(80);
	sAlarm3: STRING(80);
	sAlarm4: STRING(80);
	sAlarm5: STRING(80) ;
	ifAlarmMoveStep: INT;
	bfReset: BOOL;
	ifAlarmStepClear: INT;
	bClearAlarm: BOOL;
	bDoIndex: BOOL;
	R_TRIG1: R_TRIG;
	Berror: BOOL;




	bRetIUniitAHomeNok: BOOL;
	bRetreivalUnitHomNok: BOOL;
	bRetIUniitBHomeNok: BOOL;
END_VAR
(*============Reteival Unit Error Messages================== *)


	IF bAutoModeOn AND bMCStartInAuto AND bIUnitA_StartPB AND NOT bIUnitA_RowStopperHome AND NOT bUnitARowStopperStarted  THEN bRetIUniitAHomeNok:=TRUE; ELSE  bRetIUniitAHomeNok:=FALSE; END_IF

	IF bAutoModeOn AND bMCStartInAuto AND bIUnitB_StartPB AND NOT bIUnitB_RowStopperHome AND NOT bUnitBRowStopperStarted THEN bRetIUniitBHomeNok:=TRUE; ELSE  bRetIUniitBHomeNok:=FALSE; END_IF

	IF bRetIUniitAHomeNok OR bRetIUniitAHomeNok THEN bRetreivalUnitHomNok:=TRUE; ELSE bRetreivalUnitHomNok:=FALSE; END_IF


















(*

IF bfAlarmbit1 THEN sAlarmBuffer[1]:=sAlarm1;bfAlarmbit1:=FALSE; END_IF
IF bfAlarmbit2 THEN sAlarmBuffer[2]:=sAlarm2;bfAlarmbit2:=FALSE; END_IF
IF bfAlarmbit3 THEN sAlarmBuffer[3]:=sAlarm3;bfAlarmbit3:=FALSE; END_IF
IF bfAlarmbit4 THEN sAlarmBuffer[4]:=sAlarm4;bfAlarmbit4:=FALSE; END_IF
IF bfAlarmbit5 THEN sAlarmBuffer[5]:=sAlarm5;bfAlarmbit5:=FALSE; END_IF
*)
CASE ifAlarmMoveStep OF

	0:	IF sAlarmBuffer[1]<>'' THEN ifAlarmMoveStep:=1;
			ELSIF sAlarmBuffer[2]<>'' THEN ifAlarmMoveStep:=3;
			ELSIF sAlarmBuffer[3]<>'' THEN ifAlarmMoveStep:=5;
			ELSIF sAlarmBuffer[4]<>'' THEN ifAlarmMoveStep:=7;
			ELSIF sAlarmBuffer[5]<>'' THEN ifAlarmMoveStep:=9;
		END_IF

	1:	sAlarmValue:=sAlarmBuffer[1];bfAlarmGenerated:=TRUE;ifAlarmMoveStep:=ifAlarmMoveStep+1;

	2:	IF NOT bfAlarmGenerated AND NOT bfAlarmbit1 THEN sAlarm1:=sAlarmBuffer[1]:='';ifAlarmMoveStep:=0; END_IF

	3:	sAlarmValue:=sAlarmBuffer[2];bfAlarmGenerated:=TRUE;ifAlarmMoveStep:=ifAlarmMoveStep+1;

	4:	IF NOT bfAlarmGenerated THEN sAlarm2:=sAlarmBuffer[2]:='';ifAlarmMoveStep:=0; END_IF

	5:	sAlarmValue:=sAlarmBuffer[3];bfAlarmGenerated:=TRUE;ifAlarmMoveStep:=ifAlarmMoveStep+1;

	6:	IF NOT bfAlarmGenerated THEN sAlarm3:=sAlarmBuffer[3]:='';ifAlarmMoveStep:=0; END_IF

	7:	sAlarmValue:=sAlarmBuffer[4];bfAlarmGenerated:=TRUE;ifAlarmMoveStep:=ifAlarmMoveStep+1;

	8:	IF NOT bfAlarmGenerated THEN sAlarm4:=sAlarmBuffer[4]:='';ifAlarmMoveStep:=0; END_IF

	9:	sAlarmValue:=sAlarmBuffer[5];bfAlarmGenerated:=TRUE;ifAlarmMoveStep:=ifAlarmMoveStep+1;

	10:	IF NOT bfAlarmGenerated THEN sAlarm5:=sAlarmBuffer[5]:='';ifAlarmMoveStep:=0; END_IF

END_CASE






IF bfAlarmGenerated THEN
CASE ifAlarmStep OF

	0: 	k:=50;ifAlarmStep:=ifAlarmStep+1;

	1:	sAlarmArray[k]:=sAlarmArray[k-1];ifAlarmStep:=ifAlarmStep+1;

	2: 	IF NOT (k=1) THEN k:=k-1;ifAlarmStep:=1; ELSE ifAlarmStep:=ifAlarmStep+1; END_IF

	3:	sAlarmArray[0]:=sAlarmValue;ifAlarmStep:=ifAlarmStep+1;

	4:	bfAlarmGenerated:=FALSE;ifAlarmStep:=0;

END_CASE
END_IF
(*
 IF bClearAlarm THEN
FOR i:=0 TO 50 DO
	sAlarmArray[i]:='';
END_FOR
END_IF
*)
IF bFeedinfCylFwdRsError THEN sAlarmBuffer[1]:='chect Cone Feeding Piston Fwd Reed Switdh'; ELSE sAlarmBuffer[1]:=''; END_IF
IF bfAlarmbit2 THEN sAlarmBuffer[2]:=sAlarm2;ELSE sAlarmBuffer[2]:=''; END_IF
IF bfAlarmbit3 THEN sAlarmBuffer[3]:=sAlarm3;ELSE sAlarmBuffer[3]:=''; END_IF
IF bfAlarmbit4 THEN sAlarmBuffer[4]:=sAlarm4;ELSE sAlarmBuffer[4]:=''; END_IF
IF bfAlarmbit5 THEN sAlarmBuffer[5]:=sAlarm5;ELSE sAlarmBuffer[5]:=''; END_IF

IF bfAlarmbit1 OR bfAlarmbit2 OR bfAlarmbit3 OR bfAlarmbit4 OR bfAlarmbit5 THEN
Berror:=TRUE;
ELSE
Berror:=FALSE;
END_IF
END_PROGRAM

(* POU Auto/Gripper/SDOREAD, CFC *)
PROGRAM SDOREAD
VAR
	rd1: ADSREAD;
		TON1: TON;
	testx: BOOL;
	WRI1: ADSWRITE;

	testy: BOOL;
	rd2: ADSREAD;
	testz: BOOL;
	rd3: ADSREAD;
	CurrAct: INT;
	ReadCurrent: BOOL;
	WRI2: ADSWRITE;
	HomeMethod: BYTE;
	bWrHomeMethod: BOOL;
	Rd4: ADSREAD;
	TMtimer: TON;
	patIMER: TON;
	rd5: ADSREAD;
	VeloAct: DINT;
	VATimer: TON;
	ReadTargetVelo: BOOL;
	VeloSet: DINT;
	rd6: ADSREAD;
	Write3: ADSWRITE;
	TVWTimer: TON;
	WRI4: ADSWRITE;
	Rd7: ADSREAD;
	ReadActTorq: BOOL;
	testbit: BOOL;
	TorqueRead: ADSREAD;
	bAModeWritetemp: BOOL;
	testPer: FB_WritePersistentData;
	WRI10: ADSWRITE;
	BSample: BOOL;
	Rd8: ADSREAD;
	Denom: INT;
	timer10: TON;
	wr9: ADSWRITE;
	Denomwr: INT:=1000;
	timer11: TON;
END_VAR
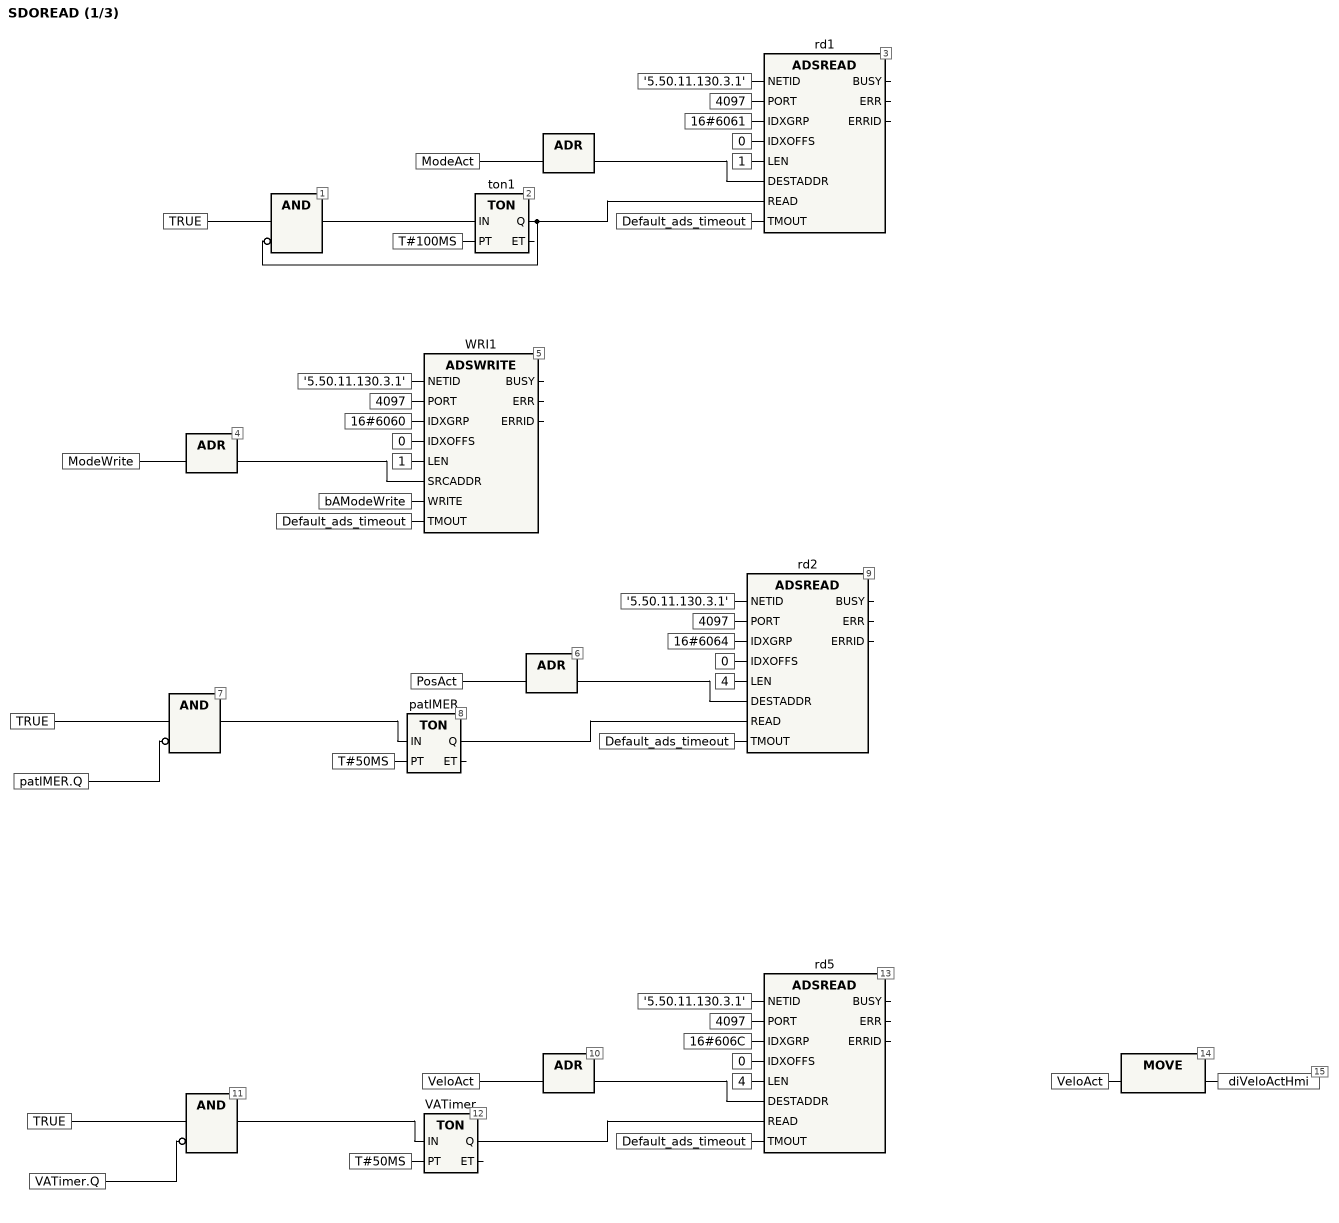
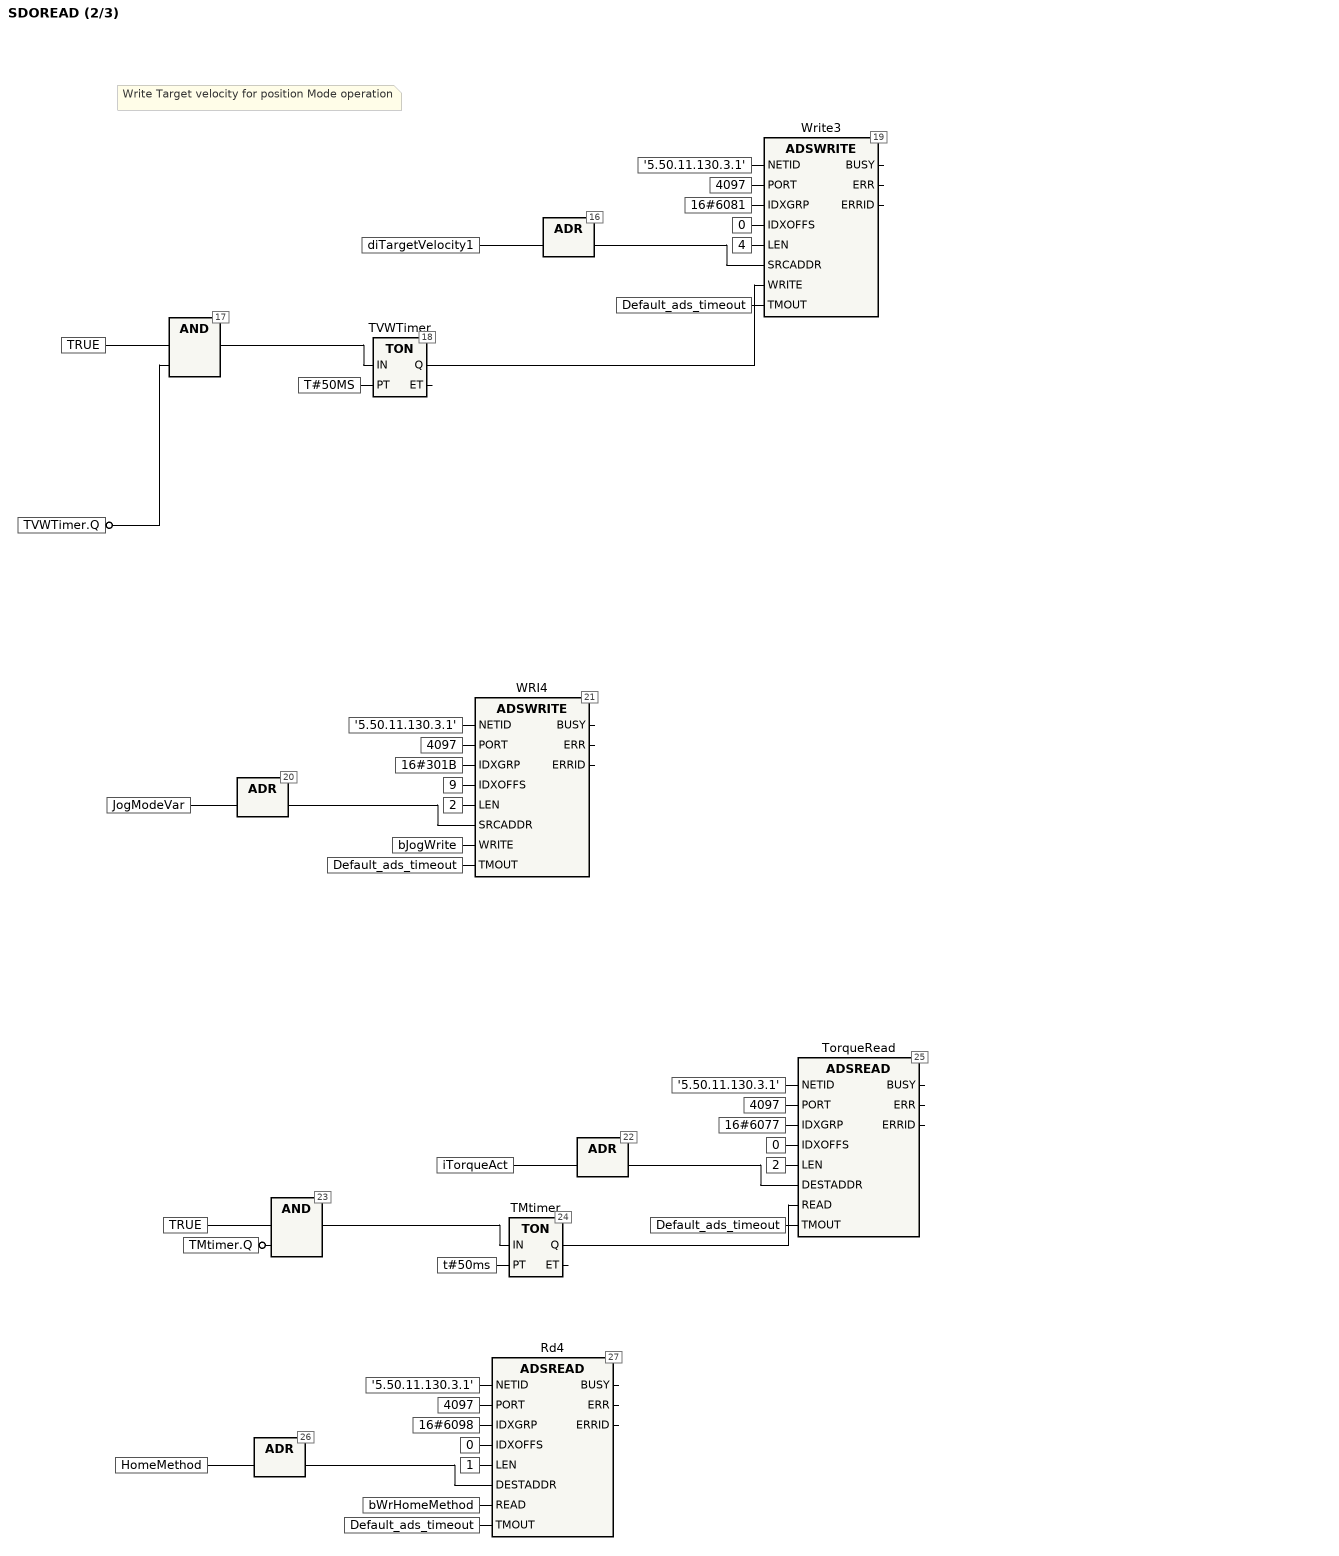
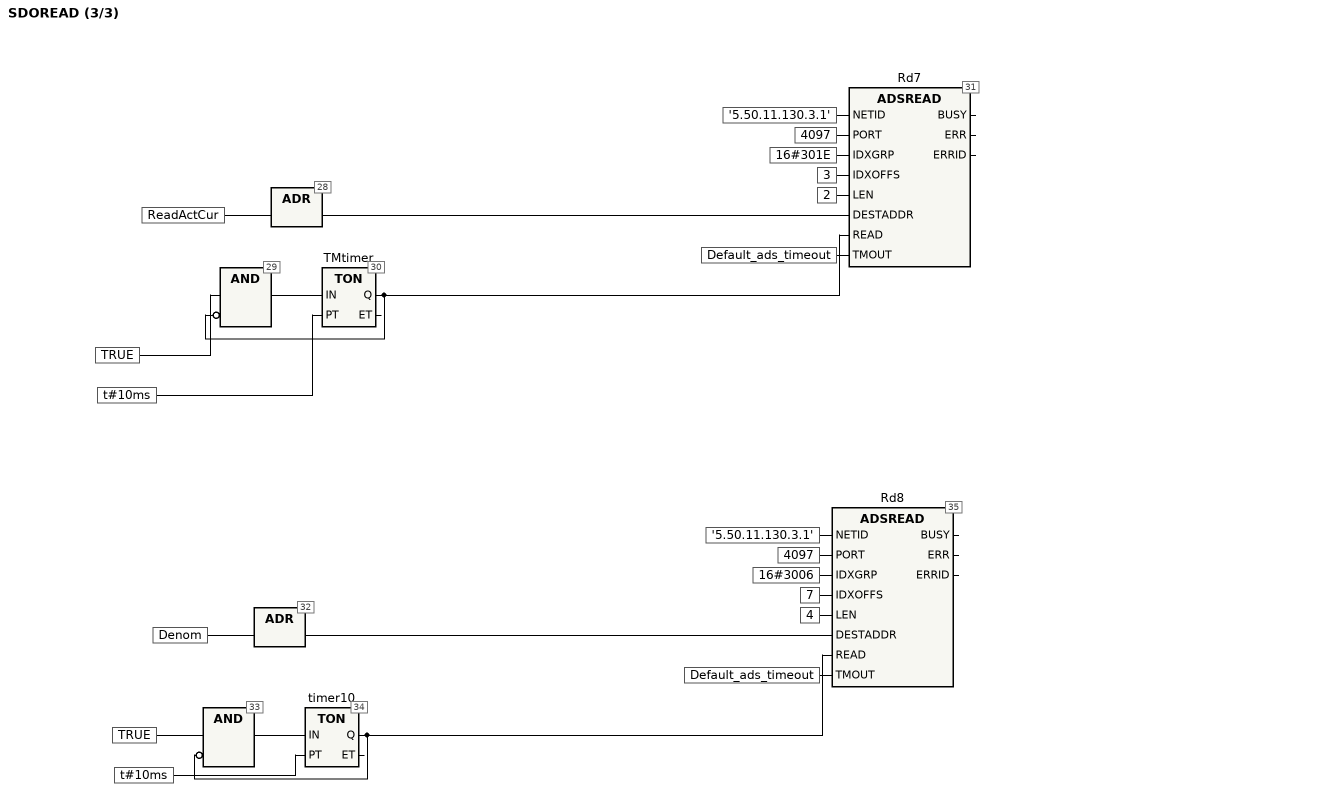
_CFC_ (* Continuous Function Chart, elements in execution order *)
(* Write Target velocity for position Mode operation *)
#0 ADR(ModeAct)
#1 AND(TRUE, NOT #2.Q)
#2 ton1:TON(IN: #1, PT: T#100MS)
#3 rd1:ADSREAD(NETID: '5.50.11.130.3.1', PORT: 4097, IDXGRP: 16#6061, IDXOFFS: 0, LEN: 1, DESTADDR: #0, READ: #2.Q, TMOUT: Default_ads_timeout)
#4 ADR(ModeWrite)
#5 WRI1:ADSWRITE(NETID: '5.50.11.130.3.1', PORT: 4097, IDXGRP: 16#6060, IDXOFFS: 0, LEN: 1, SRCADDR: #4, WRITE: bAModeWrite, TMOUT: Default_ads_timeout)
#6 ADR(PosAct)
#7 AND(TRUE, NOT patIMER.Q)
#8 patIMER:TON(IN: #7, PT: T#50MS)
#9 rd2:ADSREAD(NETID: '5.50.11.130.3.1', PORT: 4097, IDXGRP: 16#6064, IDXOFFS: 0, LEN: 4, DESTADDR: #6, READ: #8.Q, TMOUT: Default_ads_timeout)
#10 ADR(VeloAct)
#11 AND(TRUE, NOT VATimer.Q)
#12 VATimer:TON(IN: #11, PT: T#50MS)
#13 rd5:ADSREAD(NETID: '5.50.11.130.3.1', PORT: 4097, IDXGRP: 16#606C, IDXOFFS: 0, LEN: 4, DESTADDR: #10, READ: #12.Q, TMOUT: Default_ads_timeout)
#14 MOVE(VeloAct)
#15 diVeloActHmi <= #14
#16 ADR(diTargetVelocity1)
#17 AND(TRUE, NOT TVWTimer.Q)
#18 TVWTimer:TON(IN: #17, PT: T#50MS)
#19 Write3:ADSWRITE(NETID: '5.50.11.130.3.1', PORT: 4097, IDXGRP: 16#6081, IDXOFFS: 0, LEN: 4, SRCADDR: #16, WRITE: #18.Q, TMOUT: Default_ads_timeout)
#20 ADR(JogModeVar)
#21 WRI4:ADSWRITE(NETID: '5.50.11.130.3.1', PORT: 4097, IDXGRP: 16#301B, IDXOFFS: 9, LEN: 2, SRCADDR: #20, WRITE: bJogWrite, TMOUT: Default_ads_timeout)
#22 ADR(iTorqueAct)
#23 AND(TRUE, NOT TMtimer.Q)
#24 TMtimer:TON(IN: #23, PT: t#50ms)
#25 TorqueRead:ADSREAD(NETID: '5.50.11.130.3.1', PORT: 4097, IDXGRP: 16#6077, IDXOFFS: 0, LEN: 2, DESTADDR: #22, READ: #24.Q, TMOUT: Default_ads_timeout)
#26 ADR(HomeMethod)
#27 Rd4:ADSREAD(NETID: '5.50.11.130.3.1', PORT: 4097, IDXGRP: 16#6098, IDXOFFS: 0, LEN: 1, DESTADDR: #26, READ: bWrHomeMethod, TMOUT: Default_ads_timeout)
#28 ADR(ReadActCur)
#29 AND(TRUE, NOT #30.Q)
#30 TMtimer:TON(IN: #29, PT: t#10ms)
#31 Rd7:ADSREAD(NETID: '5.50.11.130.3.1', PORT: 4097, IDXGRP: 16#301E, IDXOFFS: 3, LEN: 2, DESTADDR: #28, READ: #30.Q, TMOUT: Default_ads_timeout)
#32 ADR(Denom)
#33 AND(TRUE, NOT #34.Q)
#34 timer10:TON(IN: #33, PT: t#10ms)
#35 Rd8:ADSREAD(NETID: '5.50.11.130.3.1', PORT: 4097, IDXGRP: 16#3006, IDXOFFS: 7, LEN: 4, DESTADDR: #32, READ: #34.Q, TMOUT: Default_ads_timeout)
_END_CFC_
(* the same logic as Structured Text *)
(* Write Target velocity for position Mode operation *)
ton1(IN := TRUE AND NOT ton1.Q, PT := T#100MS);
rd1(NETID := '5.50.11.130.3.1', PORT := 4097, IDXGRP := 16#6061, IDXOFFS := 0, LEN := 1, DESTADDR := ADR(ModeAct), READ := ton1.Q, TMOUT := Default_ads_timeout);
WRI1(NETID := '5.50.11.130.3.1', PORT := 4097, IDXGRP := 16#6060, IDXOFFS := 0, LEN := 1, SRCADDR := ADR(ModeWrite), WRITE := bAModeWrite, TMOUT := Default_ads_timeout);
patIMER(IN := TRUE AND NOT patIMER.Q, PT := T#50MS);
rd2(NETID := '5.50.11.130.3.1', PORT := 4097, IDXGRP := 16#6064, IDXOFFS := 0, LEN := 4, DESTADDR := ADR(PosAct), READ := patIMER.Q, TMOUT := Default_ads_timeout);
VATimer(IN := TRUE AND NOT VATimer.Q, PT := T#50MS);
rd5(NETID := '5.50.11.130.3.1', PORT := 4097, IDXGRP := 16#606C, IDXOFFS := 0, LEN := 4, DESTADDR := ADR(VeloAct), READ := VATimer.Q, TMOUT := Default_ads_timeout);
diVeloActHmi := VeloAct;
TVWTimer(IN := TRUE AND NOT TVWTimer.Q, PT := T#50MS);
Write3(NETID := '5.50.11.130.3.1', PORT := 4097, IDXGRP := 16#6081, IDXOFFS := 0, LEN := 4, SRCADDR := ADR(diTargetVelocity1), WRITE := TVWTimer.Q, TMOUT := Default_ads_timeout);
WRI4(NETID := '5.50.11.130.3.1', PORT := 4097, IDXGRP := 16#301B, IDXOFFS := 9, LEN := 2, SRCADDR := ADR(JogModeVar), WRITE := bJogWrite, TMOUT := Default_ads_timeout);
TMtimer(IN := TRUE AND NOT TMtimer.Q, PT := t#50ms);
TorqueRead(NETID := '5.50.11.130.3.1', PORT := 4097, IDXGRP := 16#6077, IDXOFFS := 0, LEN := 2, DESTADDR := ADR(iTorqueAct), READ := TMtimer.Q, TMOUT := Default_ads_timeout);
Rd4(NETID := '5.50.11.130.3.1', PORT := 4097, IDXGRP := 16#6098, IDXOFFS := 0, LEN := 1, DESTADDR := ADR(HomeMethod), READ := bWrHomeMethod, TMOUT := Default_ads_timeout);
TMtimer(IN := TRUE AND NOT TMtimer.Q, PT := t#10ms);
Rd7(NETID := '5.50.11.130.3.1', PORT := 4097, IDXGRP := 16#301E, IDXOFFS := 3, LEN := 2, DESTADDR := ADR(ReadActCur), READ := TMtimer.Q, TMOUT := Default_ads_timeout);
timer10(IN := TRUE AND NOT timer10.Q, PT := t#10ms);
Rd8(NETID := '5.50.11.130.3.1', PORT := 4097, IDXGRP := 16#3006, IDXOFFS := 7, LEN := 4, DESTADDR := ADR(Denom), READ := timer10.Q, TMOUT := Default_ads_timeout);
END_PROGRAM

(* Visualisation AA
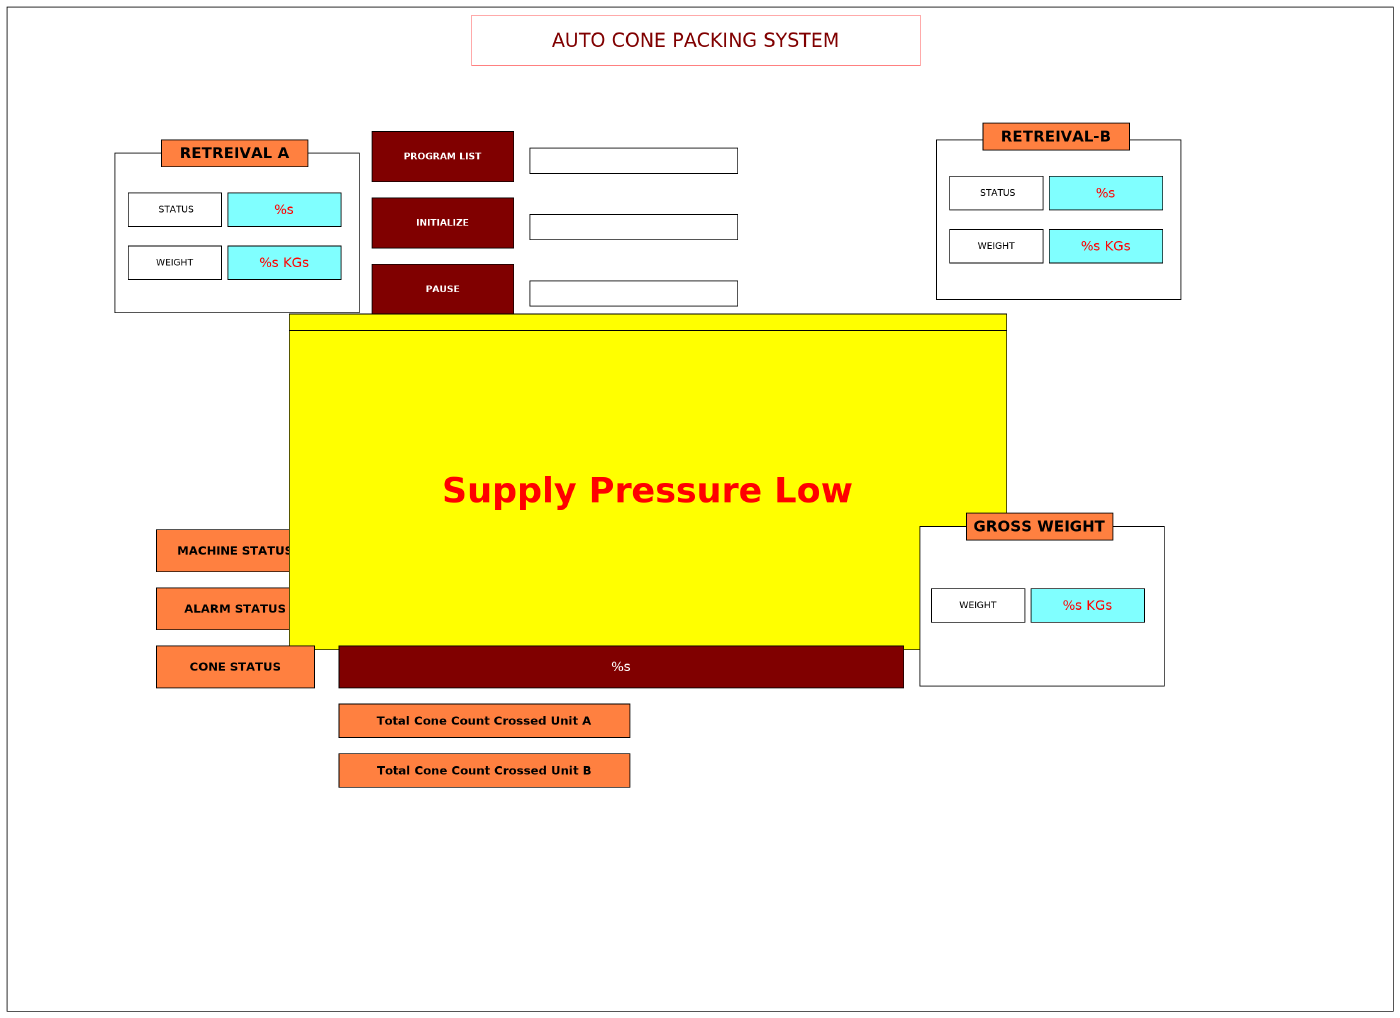
rounded rectangle at (440,140)-(611,201): text "PROGRAM LIST"; opens Models
rounded rectangle at (440,220)-(611,281): text "INITIALIZE"; alarm colour if bAInitializeSeq; taps bInitializeHmi
rounded rectangle at (440,470)-(611,531): text "STOP"; alarm colour if bStopHmi; taps bStopHmi
rounded rectangle at (630,160)-(881,191): text "PROGRAM NO"
rounded rectangle at (630,240)-(881,271): text "DETAILS"
rounded rectangle at (630,320)-(881,351): text "NO OF CONE PROCESSED"
rounded rectangle at (630,400)-(881,431): text "NO OF CARTONS PROCESSED"
rounded rectangle at (630,480)-(881,511): text "DATE"
rounded rectangle at (560,0)-(1101,61): text "AUTO CONE PACKING SYSTEM"
rounded rectangle at (440,300)-(611,361): text "PAUSE"; alarm colour if bAPauseSeq; taps bPauseHmi
rounded rectangle at (440,380)-(611,441): text "RESUME"; alarm colour if bAPauseSeq; taps bResumeHmi
rounded rectangle at (180,620)-(371,671): text "MACHINE STATUS"
rounded rectangle at (180,690)-(371,741): text "ALARM STATUS"
rounded rectangle at (400,690)-(1081,741): text "%s"; shows sMianAlarmStatus
group at (460,400)-(1051,611)
  rounded rectangle at (0,0)-(591,211): invisible if not bHidePopUp
  rounded rectangle at (140,110)-(251,161): text "YES"; invisible if NOT bHidePopUp; taps bPauseYesHmi
  rounded rectangle at (320,110)-(431,161): text "NO"; invisible if not bHidePopUp; taps bPauseNoHmi
  rounded rectangle at (88,16)-(513,73): text "Machine is Running. Do You Want to Change / Mode to Manual ?"; invisible if NOT bHidePopUp
  rounded rectangle at (48,168)-(553,201): text "NOTE:- All the Operations will be Aborted."; invisible if NOT bHidePopUp
rounded rectangle at (400,620)-(1081,671): text "%s"; shows sMCStatus
rounded rectangle at (340,360)-(1205,745): text "Emergency Pressed"; invisible if NOT bAEmergencyPressed
rounded rectangle at (340,380)-(1205,765): text "Supply Pressure Low"; invisible if NOT bASupplyPressureError
rounded rectangle at (400,830)-(751,871): text "Total Cone Count Crossed Unit A"
rounded rectangle at (400,890)-(751,931): text "Total Cone Count Crossed Unit B"
rounded rectangle at (180,760)-(371,811): text "CONE STATUS"
rounded rectangle at (400,760)-(1081,811): text "%s"; shows Message1_24
rounded rectangle at (630,320)-(881,351): text "NO OF CONE PROCESSED"
rounded rectangle at (630,240)-(881,271): text "DETAILS"
rounded rectangle at (630,240)-(881,271): text "DETAILS"
rounded rectangle at (630,320)-(881,351): text "NO OF CONE PROCESSED"
rounded rectangle at (630,320)-(881,351): text "NO OF CONE PROCESSED"
rounded rectangle at (630,240)-(881,271): text "DETAILS"
group at (1120,130)-(1415,343)
  rounded rectangle at (56,0)-(233,33): text "RETREIVAL-B"
  rounded rectangle at (136,64)-(273,105): text "%s"; shows sRetreivalBStatus
  rounded rectangle at (16,64)-(129,105): text "STATUS"
  rounded rectangle at (16,128)-(129,169): text "WEIGHT"
  rounded rectangle at (136,128)-(273,169): text "%s KGs"; shows .rRetUnitBWeight_Display
group at (130,150)-(425,359)
  rounded rectangle at (56,0)-(233,33): text "RETREIVAL A"
  rounded rectangle at (136,64)-(273,105): text "%s"; shows sRetreivalAStatus
  rounded rectangle at (16,64)-(129,105): text "STATUS"
  rounded rectangle at (16,128)-(129,169): text "WEIGHT"
  rounded rectangle at (136,128)-(273,169): text "%s KGs"; shows .rRetUnitAWeight_display
group at (1100,600)-(1395,809)
  rounded rectangle at (56,0)-(233,33): text "GROSS WEIGHT"
  rounded rectangle at (14,91)-(127,132): text "WEIGHT"
  rounded rectangle at (134,91)-(271,132): text "%s KGs"; shows .rGrossWeight_display
4 more shapes without text or variables
19 elements of other kinds (tables, trends, ...) not read
*)

(* Visualisation ALARM
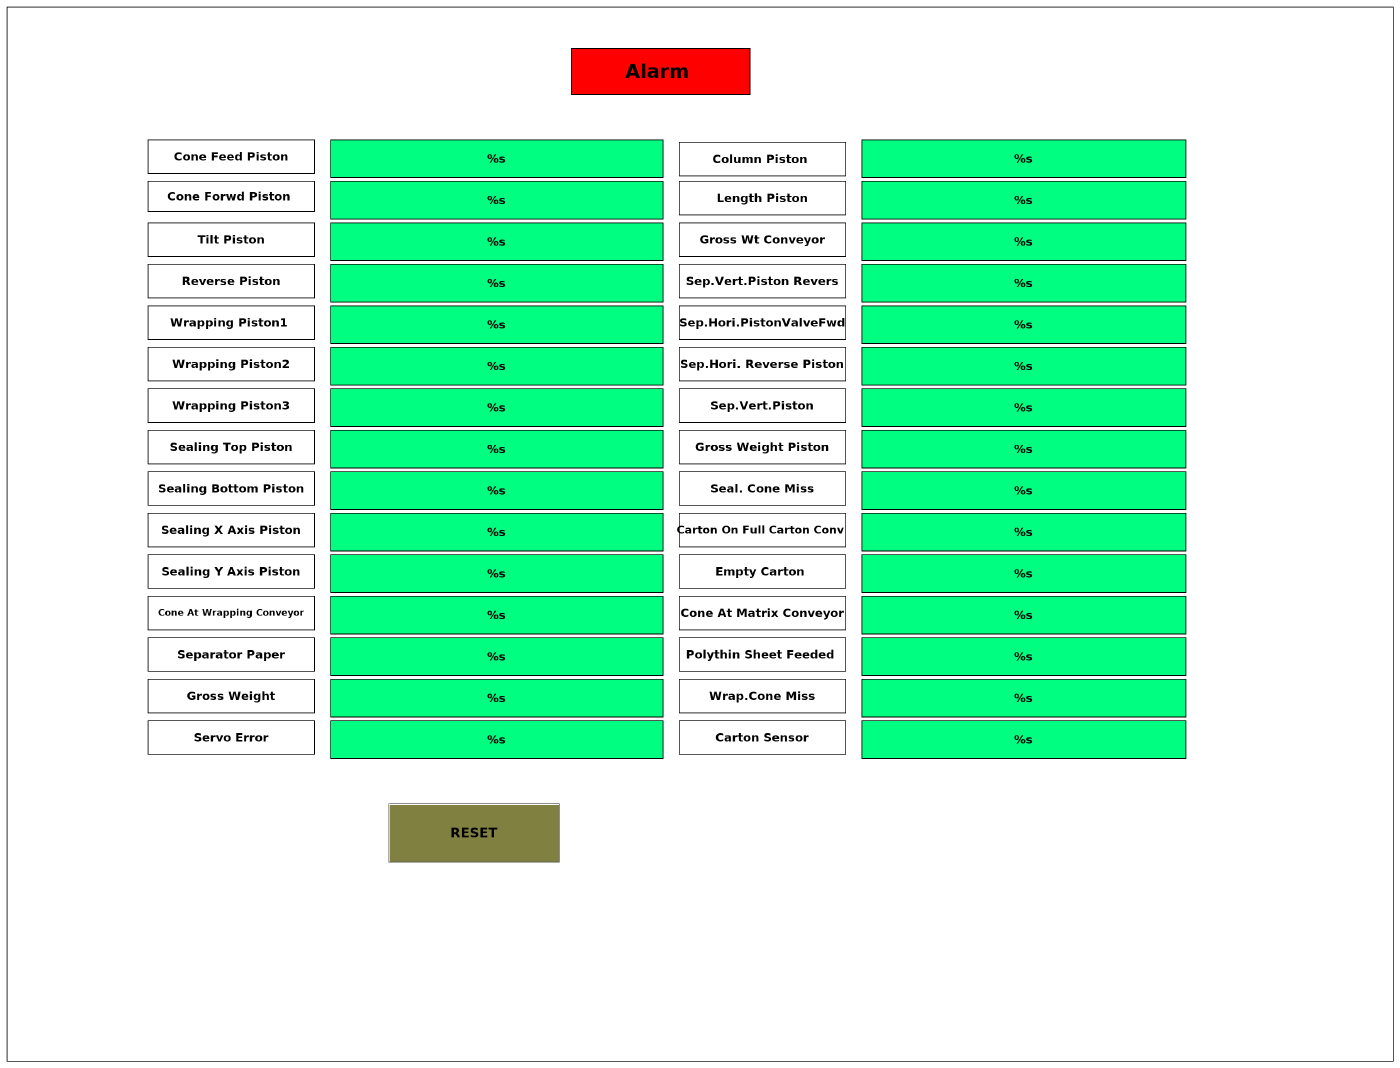
rounded rectangle at (170,200)-(371,237): text "Cone Forwd Piston"
rounded rectangle at (170,150)-(371,191): text "Cone Feed Piston"
rounded rectangle at (170,350)-(371,391): text "Wrapping Piston1"
rounded rectangle at (170,400)-(371,441): text "Wrapping Piston2"
rounded rectangle at (170,450)-(371,491): text "Wrapping Piston3"
rounded rectangle at (170,500)-(371,541): text "Sealing Top Piston"
rounded rectangle at (170,550)-(371,591): text "Sealing Bottom Piston"
rounded rectangle at (170,600)-(371,641): text "Sealing X Axis Piston"
rounded rectangle at (170,650)-(371,691): text "Sealing Y Axis Piston"
rectangle at (390,150)-(791,196): text "%s"; shows .HMIFeedPiston; alarm colour if bAConeFeddCylFwdRsError
rectangle at (390,450)-(791,496): text "%s"; shows .HMIWrapPiston3; alarm colour if bAWrap_3PistRsError
rectangle at (390,400)-(791,446): text "%s"; shows .HMIWrapPiston2; alarm colour if bAWrap_2PistRsError
rectangle at (390,500)-(791,546): text "%s"; shows .HMISealTopPiston; alarm colour if bASealTopPistRsError
rectangle at (390,600)-(791,646): text "%s"; shows .HmiXAxisPiston; alarm colour if bASealSepaX_axisRsError
rectangle at (390,550)-(791,596): text "%s"; shows .HMISealBotPiston; alarm colour if bASealBottomRsError
rectangle at (390,650)-(791,696): text "%s"; shows .HmiYAxisPiston; alarm colour if bASealSepaY_axisRsError
rectangle at (390,350)-(791,396): text "%s"; shows HMIWrapPiston1; alarm colour if bAWrap_1PistRsError
rectangle at (390,200)-(791,246): text "%s"; shows .HMIForwdPiston; alarm colour if bAForwPistRsError
rounded rectangle at (680,40)-(896,96): text "Alarm"
button at (460,950)-(666,1021): text "RESET"; shows .bErrorReset; taps .bErrorReset
rounded rectangle at (170,700)-(371,741): text "Cone At Wrapping Conveyor"
rectangle at (390,700)-(791,746): text "%s"; shows sWrapConvStatus; alarm colour if baConePtrsentAtWrapConv
rounded rectangle at (810,550)-(1011,591): text "Seal. Cone Miss"
rectangle at (1030,550)-(1421,596): text "%s"; shows .SealConeMiss; alarm colour if (SealBitAlert OR bQSealBitAlert )
rounded rectangle at (810,600)-(1011,641): text "Carton On Full Carton Conv"
rectangle at (1030,600)-(1421,646): text "%s"; shows HmiFullCartonAtConveyer; alarm colour if bHmiColourChangeBit
rounded rectangle at (810,153)-(1011,194): text "Column Piston"
rounded rectangle at (170,250)-(371,291): text "Tilt Piston"
rounded rectangle at (170,300)-(371,341): text "Reverse Piston"
rounded rectangle at (810,500)-(1011,541): text "Gross Weight Piston"
rounded rectangle at (810,400)-(1011,441): text "Sep.Hori. Reverse Piston"
rounded rectangle at (810,300)-(1011,341): text "Sep.Vert.Piston Revers"
rounded rectangle at (810,450)-(1011,491): text "Sep.Vert.Piston"
rounded rectangle at (810,350)-(1011,391): text "Sep.Hori.PistonValveFwd"
rectangle at (390,250)-(791,296): text "%s"; shows .HmiTiltPiston; alarm colour if bATiltPistRsError
rectangle at (1030,500)-(1421,546): text "%s"; shows .HmiGrossWtPiston; alarm colour if bAGrossWtSenRsError
rectangle at (390,300)-(791,346): text "%s"; shows .HmiReverPiston; alarm colour if bAReversPistnRsError
rectangle at (1030,400)-(1421,446): text "%s"; shows .HmiSepHoriRevPiston; alarm colour if bASepaHoriRevValveRsError
rectangle at (1030,450)-(1421,496): text "%s"; shows .HmiSepVertiPiston
rectangle at (1030,300)-(1421,346): text "%s"; shows .HmiSepVertiPiston; alarm colour if bASepaVertiEndPistnRsError
rectangle at (1030,350)-(1421,396): text "%s"; shows .HmiSepHoriRevPiston; alarm colour if bASepaHoriForwdEndRsError
rectangle at (1030,150)-(1421,196): text "%s"; shows .HmiColuPushrPiston; alarm colour if bAColumnPushPistnRsError
rounded rectangle at (810,200)-(1011,241): text "Length Piston"
rectangle at (1030,200)-(1421,246): text "%s"; shows .HmiLengthPiston; alarm colour if bAL_BTightHomeSenRsError
rounded rectangle at (810,250)-(1011,291): text "Gross Wt Conveyor"
rectangle at (1030,250)-(1421,296): text "%s"; shows sOneMinConMsg; alarm colour if bACartonOnGrossWtConv
rounded rectangle at (810,650)-(1011,691): text "Empty Carton"
rectangle at (1030,650)-(1421,696): text "%s"; shows HMIEmptyCartonDetectErr; alarm colour if bEmptyCartonDetectError
rounded rectangle at (810,700)-(1011,741): text "Cone At Matrix Conveyor"
rectangle at (1030,700)-(1421,746): text "%s"; shows sMatrixConvStatus; alarm colour if bAConeMissAtMatricConv
rounded rectangle at (170,750)-(371,791): text "Separator Paper"
rectangle at (390,750)-(791,796): text "%s"; shows HMISeparatorPaperDetec; alarm colour if SeparatorAlertbit
rounded rectangle at (810,750)-(1011,791): text "Polythin Sheet Feeded"
rectangle at (1030,750)-(1421,796): text "%s"; shows bSheetNotFeeded; alarm colour if bAPolythinSheetError
rounded rectangle at (170,800)-(371,841): text "Gross Weight"
rectangle at (390,800)-(791,846): text "%s"; shows GrossWtAlarm; alarm colour if bGrossWieghtNOk
rounded rectangle at (810,800)-(1011,841): text "Wrap.Cone Miss"
rectangle at (1030,800)-(1421,846): text "%s"; shows ConeMissAlarm; alarm colour if bHmiColourChangeBit2
rounded rectangle at (810,850)-(1011,891): text "Carton Sensor"
rectangle at (1030,850)-(1421,896): text "%s"; shows HmiFullCartonAtConveyer_sensor; alarm colour if bHmiColourChangeBit2_24
rectangle at (390,850)-(791,896): text "%s"; shows sServoErrMsg; alarm colour if bServoNotReady
rounded rectangle at (170,850)-(371,891): text "Servo Error"
1 more shapes without text or variables
1 elements of other kinds (tables, trends, ...) not read
*)

(* Visualisation AUTO
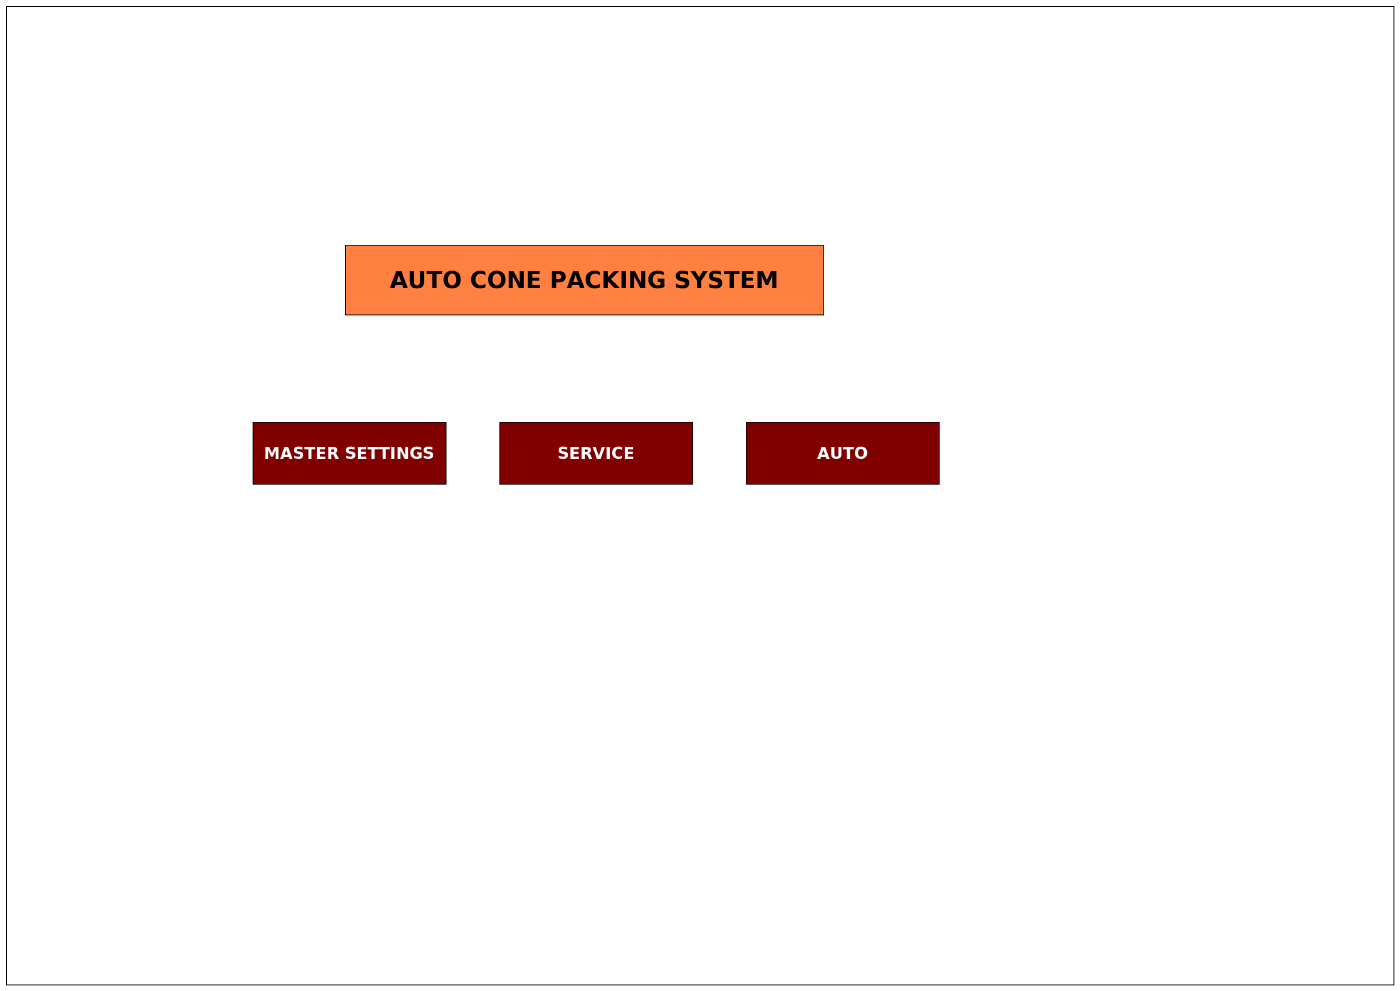
rounded rectangle at (320,540)-(571,621): text "MASTER SETTINGS"; opens MASTER_SETTINGS
rounded rectangle at (640,540)-(891,621): text "SERVICE"; opens SERVICE
rounded rectangle at (960,540)-(1211,621): text "AUTO"; opens AA
rounded rectangle at (440,310)-(1061,401): text "AUTO CONE PACKING SYSTEM"
1 more shapes without text or variables
2 elements of other kinds (tables, trends, ...) not read
*)

(* Visualisation BB
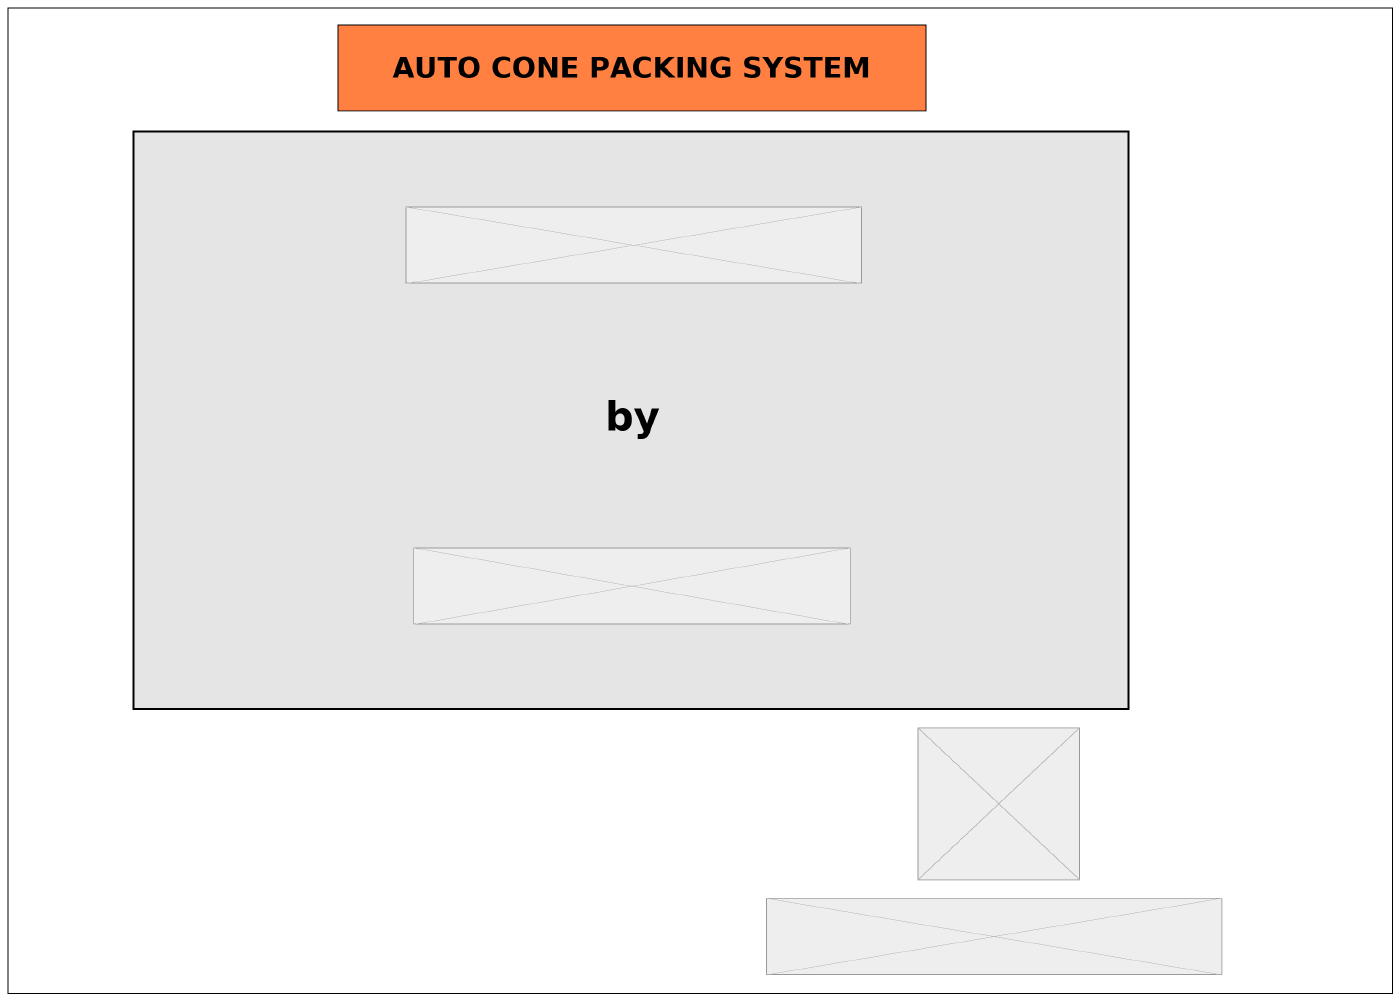
bitmap at (780,930)-(1261,1011): c:\twincat\plc\visu\autocone-logom1.jpg
rounded rectangle at (328,8)-(949,99): text "AUTO CONE PACKING SYSTEM"; invisible if NOT MAIN.EverRunTimer.Q
bitmap at (940,750)-(1111,911): c:\twincat\plc\visu\startbutton.jpg
group at (112,120)-(1169,735)
  rounded rectangle at (0,0)-(1051,611): invisible if MAIN.EverRunTimer.Q
  bitmap at (288,80)-(769,161): c:\twincat\plc\visu\autocone-logom1.jpg
  bitmap at (296,440)-(757,521): c:\twincat\plc\visu\indo_logo1.bmp
  rectangle at (272,256)-(783,347): text "by"
2 more shapes without text or variables
*)

(* Visualisation CONFIGURATION
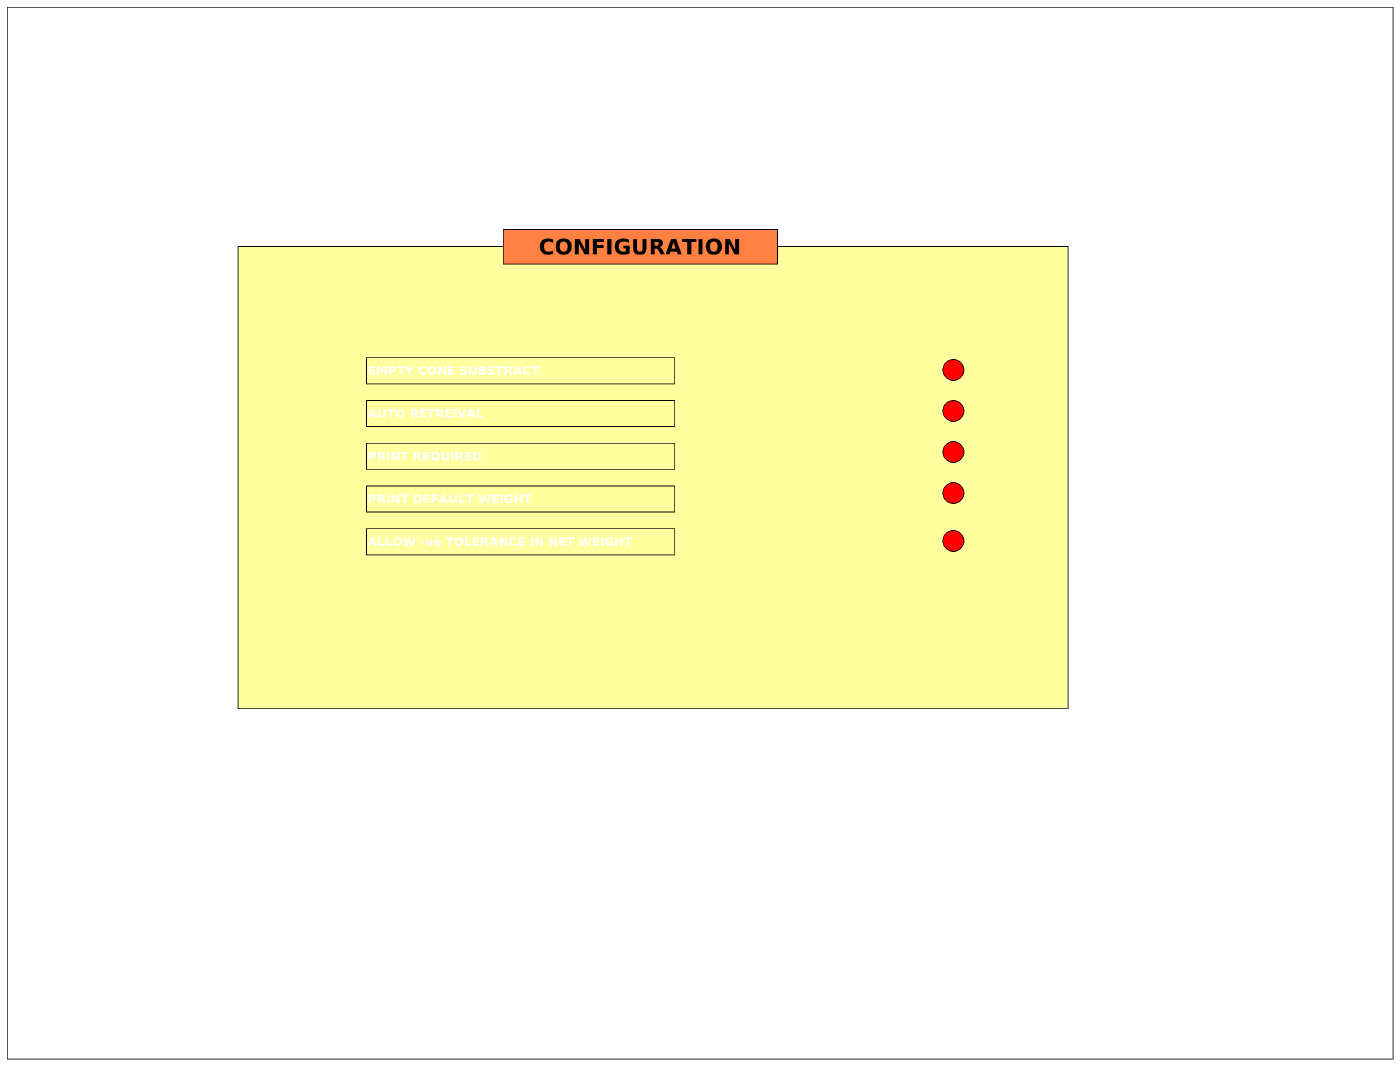
rounded rectangle at (420,410)-(781,441): text "EMPTY CONE SUBSTRACT"
rounded rectangle at (420,460)-(781,491): text "AUTO RETREIVAL"
rounded rectangle at (420,510)-(781,541): text "PRINT REQUIRED"
rounded rectangle at (420,560)-(781,591): text "PRINT DEFAULT WEIGHT"
rounded rectangle at (420,610)-(781,641): text "ALLOW -ve TOLERANCE IN NET WEIGHT"
rounded rectangle at (580,260)-(901,301): text "CONFIGURATION"
ellipse at (1094,460)-(1119,485): alarm colour if bAutoRetrivalEnabled
ellipse at (1094,412)-(1119,437): alarm colour if bEmptyConeSubEnabled
ellipse at (1094,508)-(1119,533): alarm colour if bPrintAutoEnabled
ellipse at (1094,556)-(1119,581): alarm colour if PrintDefaultWeightOnEnabled
ellipse at (1094,612)-(1119,637): alarm colour if NegToleranceEnabled
2 more shapes without text or variables
14 elements of other kinds (tables, trends, ...) not read
*)

(* Visualisation DIAGNOSTICS
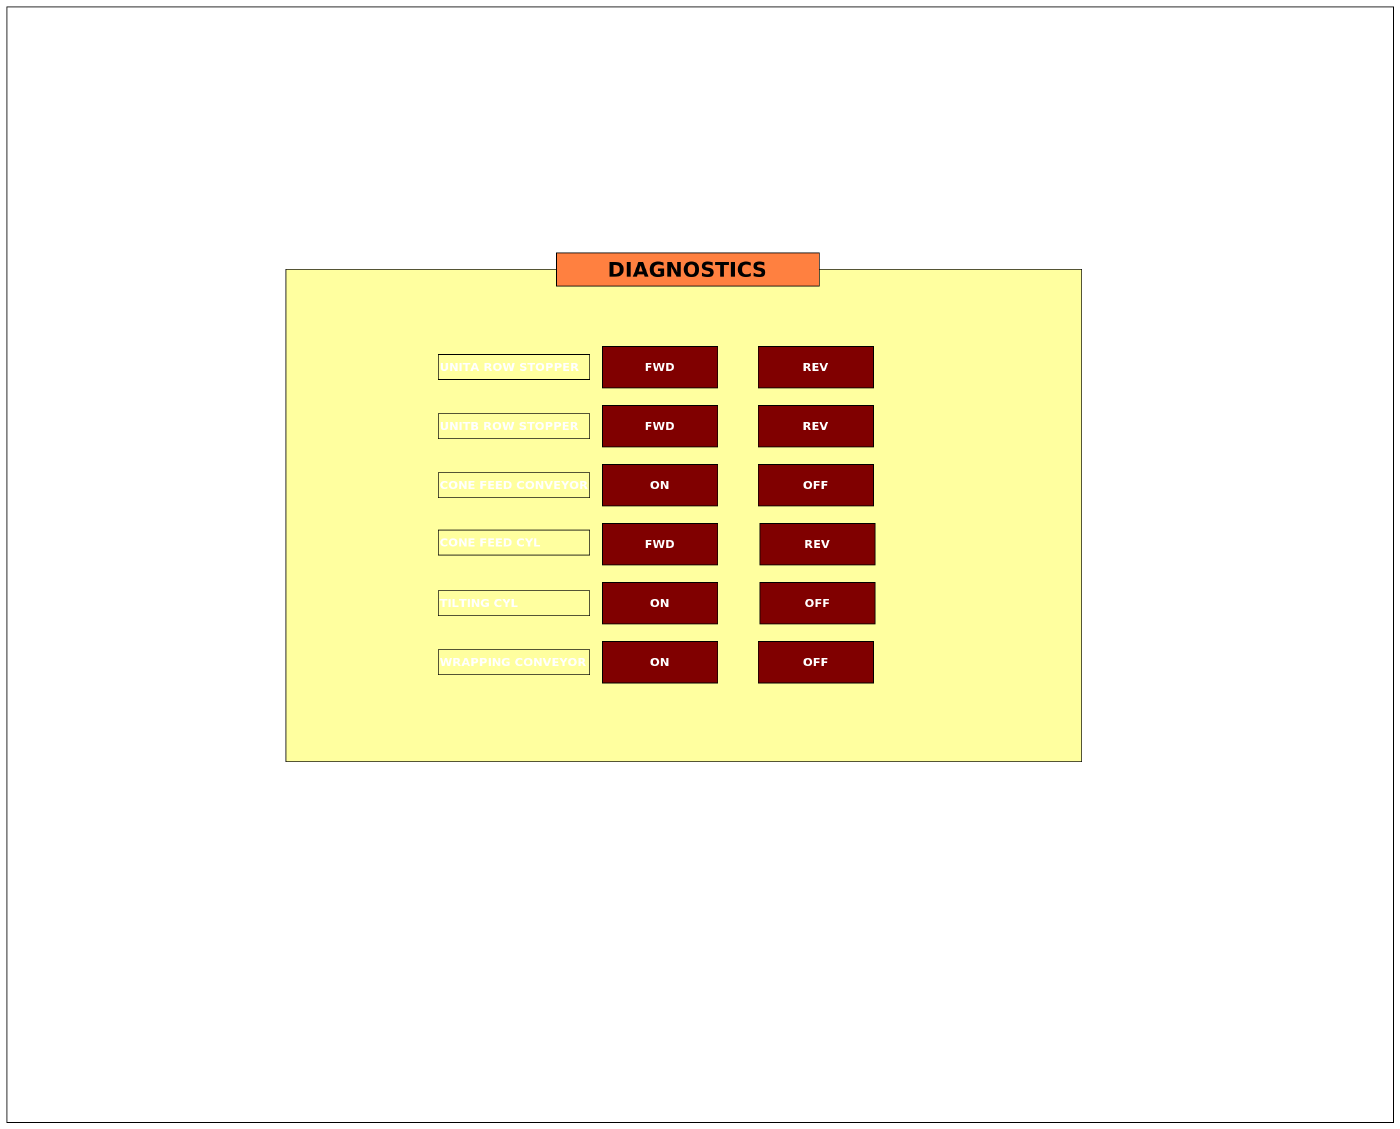
rounded rectangle at (670,210)-(991,251): text "DIAGNOSTICS"
rounded rectangle at (726,324)-(867,375): text "FWD"; alarm colour if .bUA_RowStopperMotorFwdOnHmi; taps .bUA_RowStopperMotorFwdOnHmi
rounded rectangle at (916,324)-(1057,375): text "REV"; alarm colour if .bUA_RowStopperMotorRevOnHmi; taps .bUA_RowStopperMotorRevOnHmi
rounded rectangle at (726,396)-(867,447): text "FWD"; alarm colour if .bUB_RowStopperMotorFwdOnHmi; taps .bUB_RowStopperMotorFwdOnHmi
rounded rectangle at (726,468)-(867,519): text "ON"; alarm colour if bFCMotorOnHmi; taps bFCMotorOnHmi
rounded rectangle at (916,396)-(1057,447): text "REV"; alarm colour if .bUB_RowStopperMotorRevOnHmi; taps .bUB_RowStopperMotorRevOnHmi
rounded rectangle at (916,468)-(1057,519): text "OFF"; alarm colour if bFCMotorOffHmi; taps bFCMotorOffHmi
rounded rectangle at (526,334)-(711,365): text "UNITA ROW STOPPER"
rounded rectangle at (526,406)-(711,437): text "UNITB ROW STOPPER"
rounded rectangle at (526,478)-(711,509): text "CONE FEED CONVEYOR"
rounded rectangle at (726,612)-(867,663): text "ON"; alarm colour if .bCTPistonValveOnHmi; taps .bCTPistonValveOnHmi
rounded rectangle at (918,612)-(1059,663): text "OFF"; alarm colour if .bCTPistonValveOffHmi; taps .bCTPistonValveOffHmi
rounded rectangle at (726,540)-(867,591): text "FWD"; alarm colour if .bCFPistonOnHmi; taps .bCFPistonOnHmi
rounded rectangle at (918,540)-(1059,591): text "REV"; alarm colour if .bCFPistonOffHmi; taps .bCFPistonOffHmi
rounded rectangle at (526,622)-(711,653): text "TILTING CYL"
rounded rectangle at (526,548)-(711,579): text "CONE FEED CYL"
rounded rectangle at (726,684)-(867,735): text "ON"; alarm colour if .bWCMotorOnHmi; taps .bWCMotorOnHmi
rounded rectangle at (916,684)-(1057,735): text "OFF"; alarm colour if .bWCMotorOffHmi; taps .bWCMotorOffHmi
rounded rectangle at (526,694)-(711,725): text "WRAPPING CONVEYOR"
2 more shapes without text or variables
5 elements of other kinds (tables, trends, ...) not read
*)

(* Visualisation DIAGNOSTICS_1
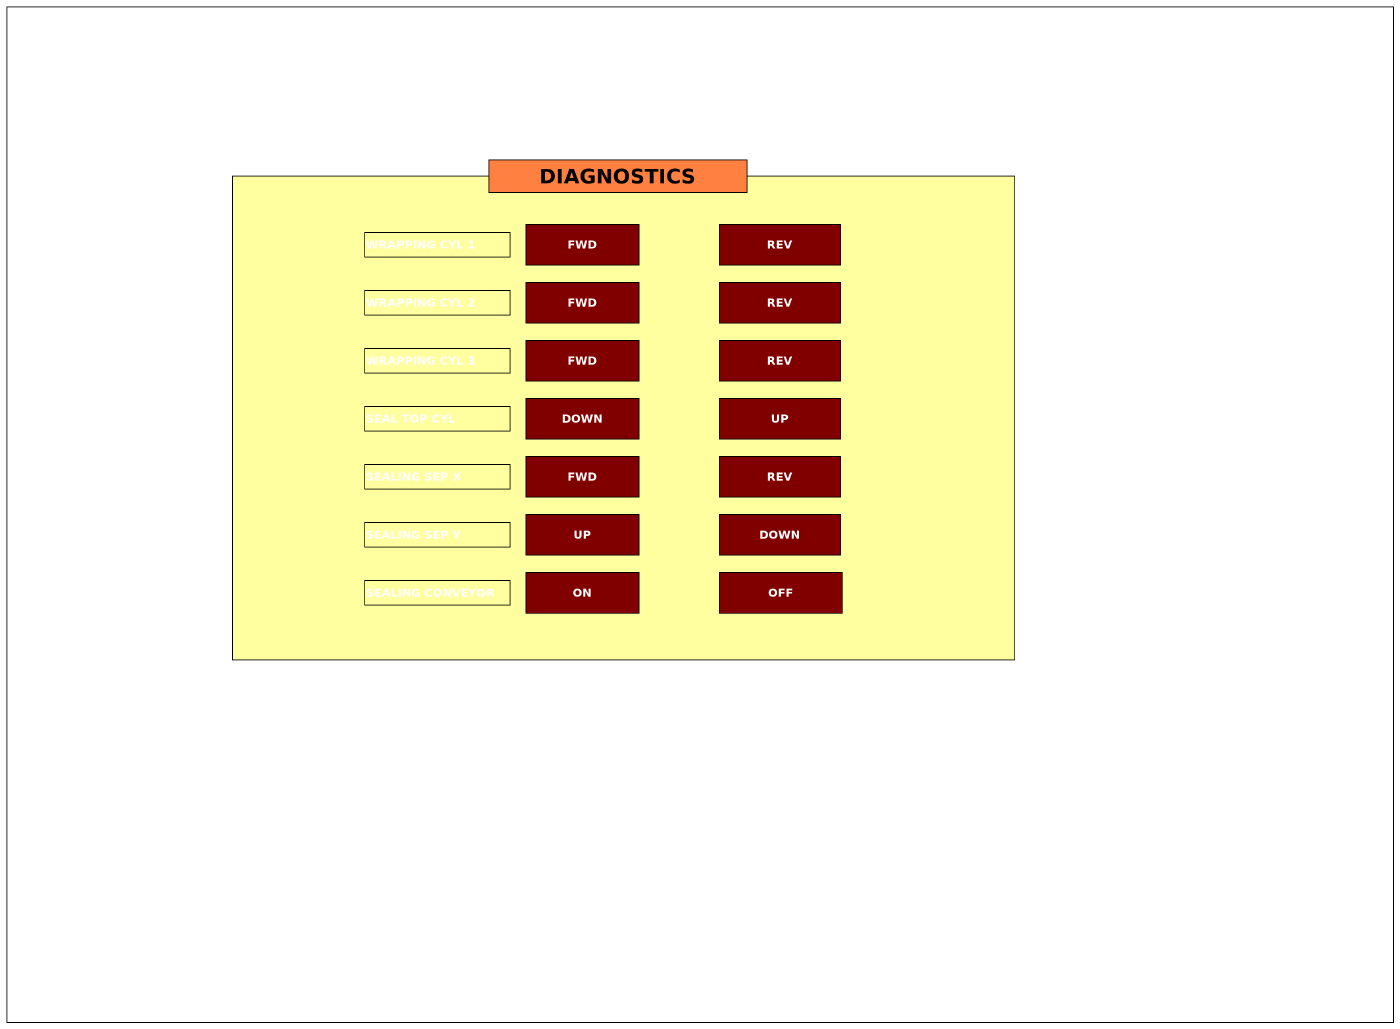
rounded rectangle at (598,190)-(919,231): text "DIAGNOSTICS"
rounded rectangle at (644,270)-(785,321): text "FWD"; alarm colour if .bWrappingCPV1OnHmi; taps .bWrappingCPV1OnHmi
rounded rectangle at (644,342)-(785,393): text "FWD"; alarm colour if .bWrappingCPV2OnHmi; taps .bWrappingCPV2OnHmi
rounded rectangle at (884,342)-(1035,393): text "REV"; alarm colour if .bWrappingCPV2OffHmi; taps .bWrappingCPV2OffHmi
rounded rectangle at (644,414)-(785,465): text "FWD"; alarm colour if .bWrappingCPV3OnHmi; taps .bWrappingCPV3OnHmi
rounded rectangle at (884,414)-(1035,465): text "REV"; alarm colour if .bWrappingCPV3OffHmi; taps .bWrappingCPV3OffHmi
rounded rectangle at (644,486)-(785,537): text "DOWN"; alarm colour if .bSealingTopPVOnHmi; taps .bSealingTopPVOnHmi
rounded rectangle at (884,486)-(1035,537): text "UP"; alarm colour if bSealingTopPVOffHmi; taps bSealingTopPVOffHmi
rounded rectangle at (644,558)-(785,609): text "FWD"; alarm colour if bSSXAxisPistonValveOnHmi; taps bSSXAxisPistonValveOnHmi
rounded rectangle at (884,558)-(1035,609): text "REV"; alarm colour if bSSXAxisPistonValveOffHmi; taps bSSXAxisPistonValveOffHmi
rounded rectangle at (444,280)-(625,311): text "WRAPPING CYL 1"
rounded rectangle at (444,352)-(625,383): text "WRAPPING CYL 2"
rounded rectangle at (444,424)-(625,455): text "WRAPPING CYL 3"
rounded rectangle at (444,496)-(625,527): text "SEAL TOP CYL"
rounded rectangle at (444,568)-(625,599): text "SEALING SEP X"
rounded rectangle at (884,270)-(1035,321): text "REV"; alarm colour if .bWrappingCPV1OffHmi; taps .bWrappingCPV1OffHmi
rounded rectangle at (644,702)-(785,753): text "ON"; alarm colour if bSCMotorOnHmi; taps bSCMotorOnHmi
rounded rectangle at (884,702)-(1037,753): text "OFF"; alarm colour if bSCMotorOffHmi; taps bSCMotorOffHmi
rounded rectangle at (444,712)-(625,743): text "SEALING CONVEYOR"
rounded rectangle at (644,630)-(785,681): text "UP"; alarm colour if bSSYAxisPistonValveOnHmi; taps bSSYAxisPistonValveOnHmi
rounded rectangle at (884,630)-(1035,681): text "DOWN"; alarm colour if bSSYAxisPistonValveOffHmi; taps bSSYAxisPistonValveOffHmi
rounded rectangle at (444,640)-(625,671): text "SEALING SEP Y"
2 more shapes without text or variables
5 elements of other kinds (tables, trends, ...) not read
*)

(* Visualisation DIAGNOSTICS_2
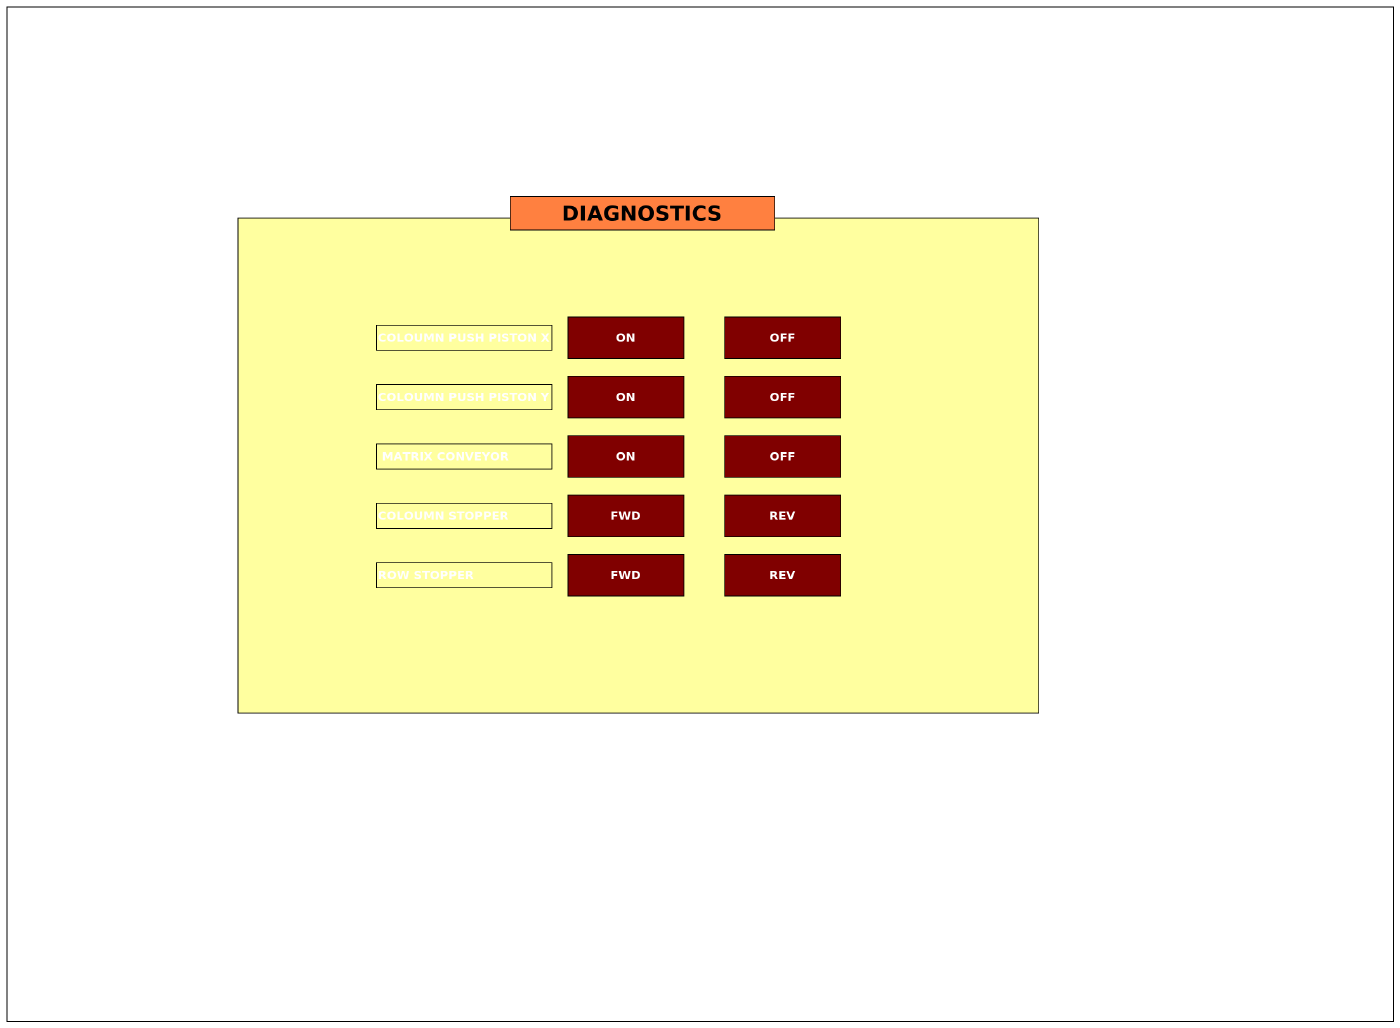
rounded rectangle at (610,230)-(931,271): text "DIAGNOSTICS"
rounded rectangle at (870,520)-(1011,571): text "OFF"; alarm colour if .bMCMotorOffHmi; taps .bMCMotorOffHmi
rounded rectangle at (680,520)-(821,571): text "ON"; alarm colour if .bMCMotorOnHmi; taps .bMCMotorOnHmi
rounded rectangle at (448,530)-(661,561): text "MATRIX CONVEYOR"
rounded rectangle at (680,376)-(821,427): text "ON"; alarm colour if bCPushPistonValveOnHmi; taps bCPushPistonValveOnHmi
rounded rectangle at (870,376)-(1011,427): text "OFF"; alarm colour if bCPushPistonValveOffHmi; taps bCPushPistonValveOffHmi
rounded rectangle at (448,386)-(661,417): text "COLOUMN PUSH PISTON X"
rounded rectangle at (680,448)-(821,499): text "ON"; alarm colour if bCPushPistonValveYOnHmi; taps bCPushPistonValveYOnHmi
rounded rectangle at (870,448)-(1011,499): text "OFF"; alarm colour if bCPushPistonValveYOffHmi; taps bCPushPistonValveYOffHmi
rounded rectangle at (448,458)-(661,489): text "COLOUMN PUSH PISTON Y"
rounded rectangle at (870,592)-(1011,643): text "REV"; alarm colour if bCSMotorRevOnHmi; taps bCSMotorRevOnHmi
rounded rectangle at (680,592)-(821,643): text "FWD"; alarm colour if bCSMotorFwdOnHmi; taps bCSMotorFwdOnHmi
rounded rectangle at (448,602)-(661,633): text "COLOUMN STOPPER"
rounded rectangle at (870,664)-(1011,715): text "REV"; alarm colour if bRSMotorRevOnHmi; taps bRSMotorRevOnHmi
rounded rectangle at (680,664)-(821,715): text "FWD"; alarm colour if bRSMotorForwardOnHmi; taps bRSMotorForwardOnHmi
rounded rectangle at (448,674)-(661,705): text "ROW STOPPER"
2 more shapes without text or variables
5 elements of other kinds (tables, trends, ...) not read
*)

(* Visualisation DIAGNOSTICS_3
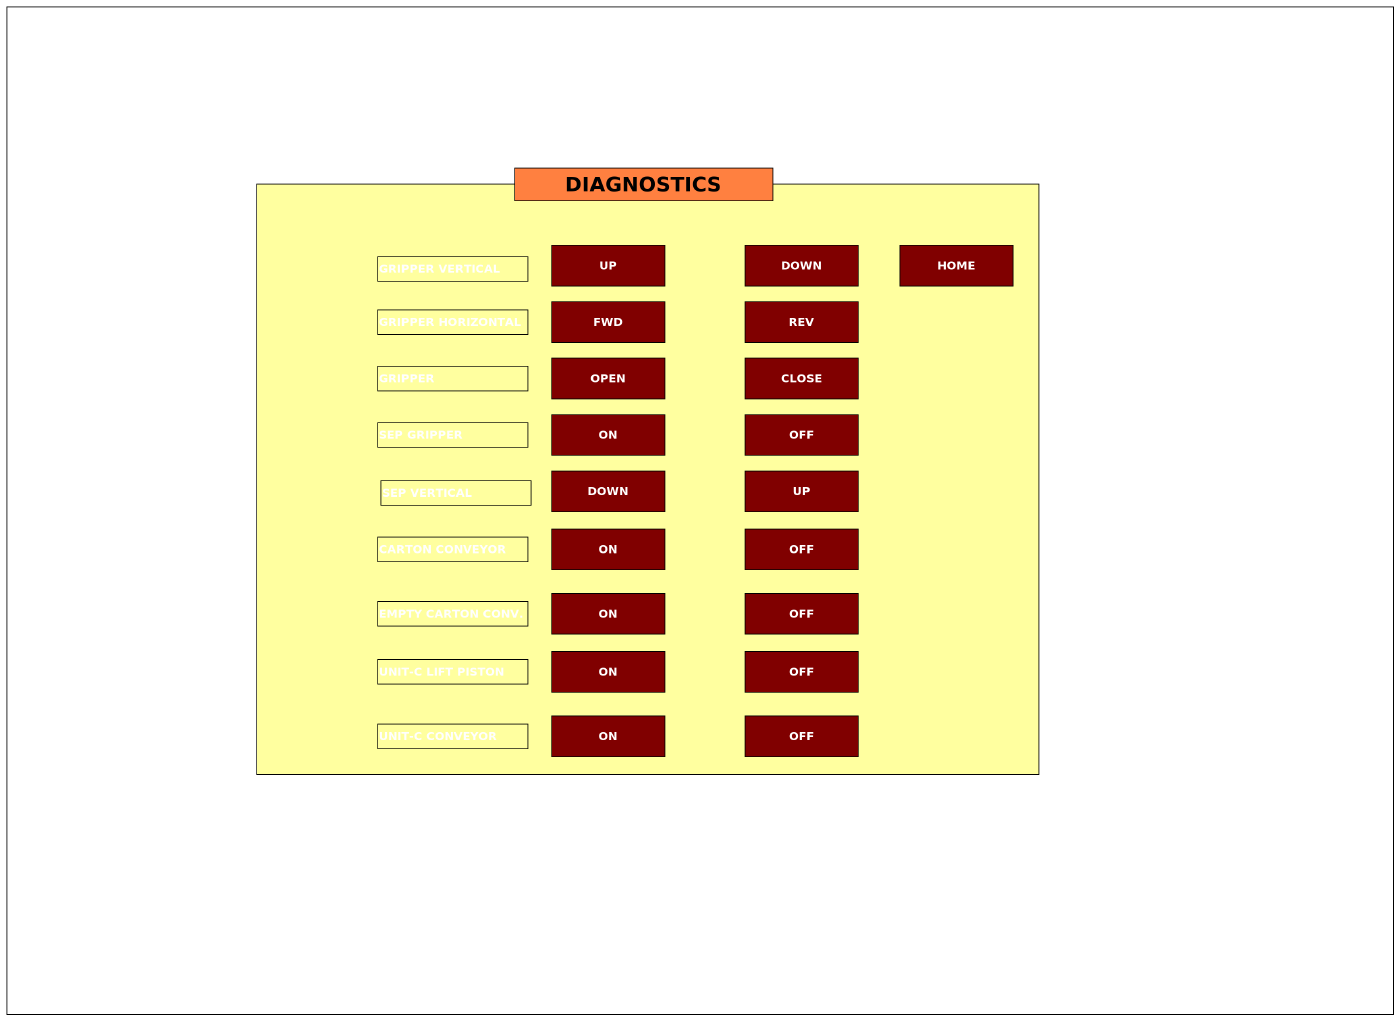
rounded rectangle at (630,180)-(951,221): text "DIAGNOSTICS"
rounded rectangle at (460,290)-(647,321): text "GRIPPER VERTICAL"
rounded rectangle at (460,356)-(647,387): text "GRIPPER HORIZONTAL"
rounded rectangle at (460,426)-(647,457): text "GRIPPER"
rounded rectangle at (460,496)-(647,527): text "SEP GRIPPER"
rounded rectangle at (676,486)-(817,537): text "ON"; alarm colour if bVPValveOnHmi; taps bVPValveOnHmi
rounded rectangle at (916,486)-(1057,537): text "OFF"; alarm colour if bVPValveOffHmi; taps bVPValveOffHmi
rounded rectangle at (676,416)-(817,467): text "OPEN"; alarm colour if .bGripperOpenHmi; taps .bGripperOpenHmi
rounded rectangle at (916,416)-(1057,467): text "CLOSE"; alarm colour if .bGrippercCloseHmi; taps .bGrippercCloseHmi
rounded rectangle at (676,346)-(817,397): text "FWD"; alarm colour if bSHPistonValveREVOnHmi; taps bSHPistonValveREVOnHmi
rounded rectangle at (916,346)-(1057,397): text "REV"; alarm colour if bSHPistonValveOnHmi; taps bSHPistonValveOnHmi
rounded rectangle at (676,276)-(817,327): text "UP"; alarm colour if bJogNegativeHmi; taps bJogNegativeHmi
rounded rectangle at (916,276)-(1057,327): text "DOWN"; alarm colour if .bJogPositiveHmi; taps .bJogPositiveHmi
rounded rectangle at (464,568)-(651,599): text "SEP VERTICAL"
rounded rectangle at (676,556)-(817,607): text "DOWN"; alarm colour if bSVPistonValveOnHmi; taps bSVPistonValveOnHmi
rounded rectangle at (916,556)-(1057,607): text "UP"; alarm colour if bSVPistonValveOffHmi; taps bSVPistonValveOffHmi
rounded rectangle at (460,638)-(647,669): text "CARTON CONVEYOR"
rounded rectangle at (676,628)-(817,679): text "ON"; alarm colour if bCCMotorOnHmi; taps bCCMotorOnHmi
rounded rectangle at (916,628)-(1057,679): text "OFF"; alarm colour if bCCMotorOffHmi; taps bCCMotorOffHmi
rounded rectangle at (460,718)-(647,749): text "EMPTY CARTON CONV."
rounded rectangle at (676,708)-(817,759): text "ON"; alarm colour if bECCMotorOnHmi; taps bECCMotorOnHmi
rounded rectangle at (916,708)-(1057,759): text "OFF"; alarm colour if bECCMotorOffHmi; taps bECCMotorOffHmi
rounded rectangle at (460,790)-(647,821): text "UNIT-C LIFT PISTON"
rounded rectangle at (676,780)-(817,831): text "ON"; alarm colour if bGWPistonOnHmi; taps bGWPistonOnHmi
rounded rectangle at (916,780)-(1057,831): text "OFF"; alarm colour if bGWPistonOffHmi1; taps bGWPistonOffHmi1
rounded rectangle at (460,870)-(647,901): text "UNIT-C CONVEYOR"
rounded rectangle at (676,860)-(817,911): text "ON"; alarm colour if bRCOnHmi; taps bRCOnHmi
rounded rectangle at (916,860)-(1057,911): text "OFF"; alarm colour if bRCOffHmi; taps bRCOffHmi
rounded rectangle at (1108,276)-(1249,327): text "HOME"; alarm colour if bServoHomeHmi; toggles bJogNegativeHmi
2 more shapes without text or variables
4 elements of other kinds (tables, trends, ...) not read
*)

(* Visualisation MASTER_SETTINGS
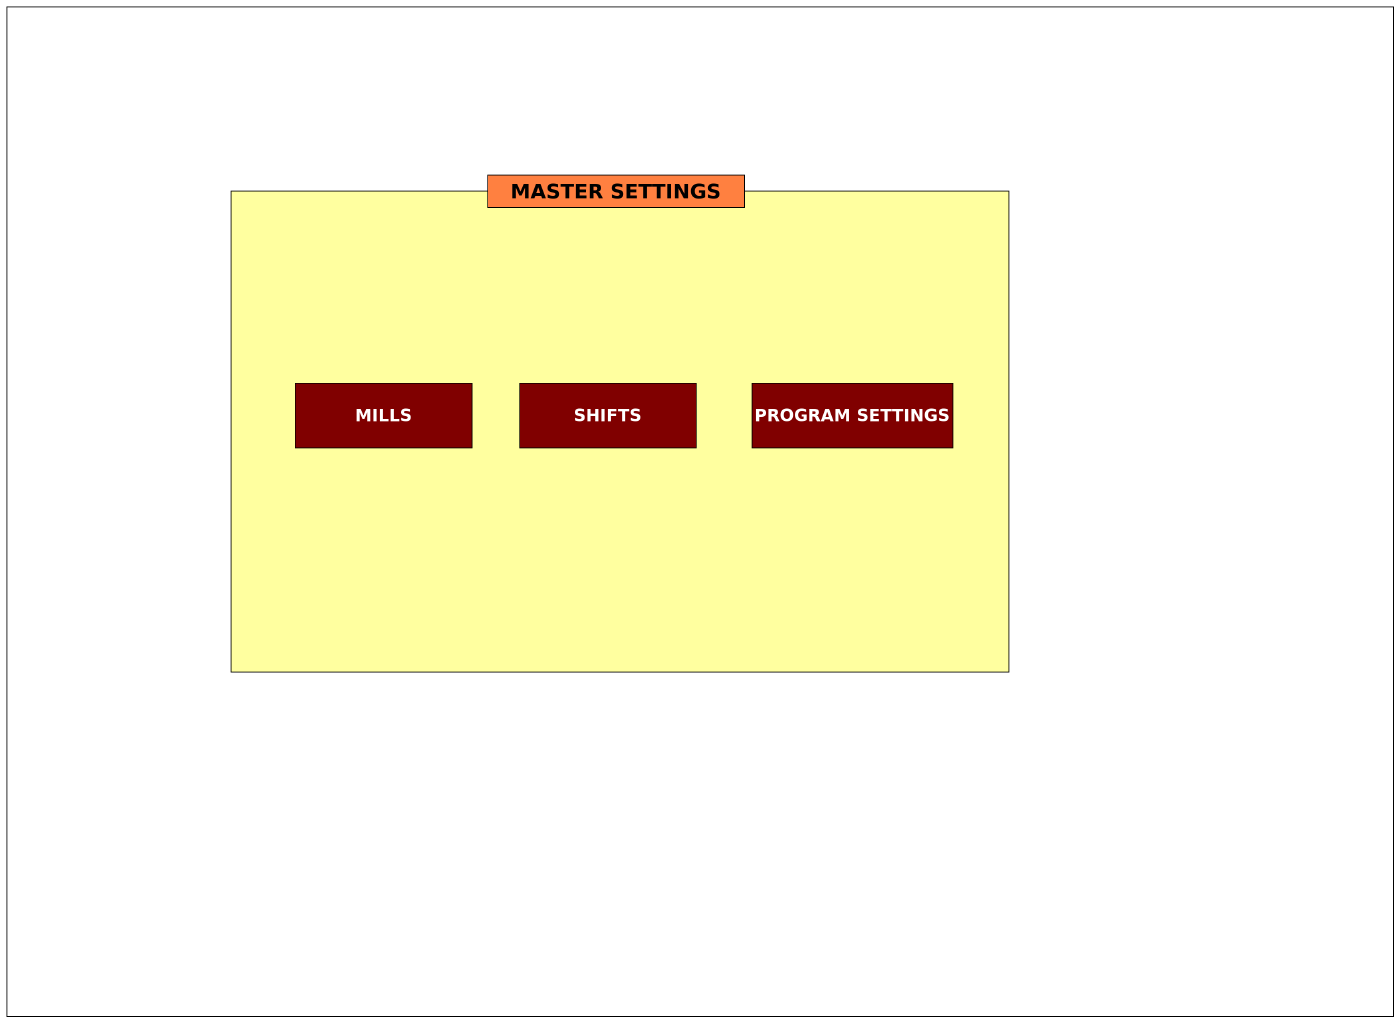
rounded rectangle at (600,210)-(921,251): text "MASTER SETTINGS"
rounded rectangle at (640,470)-(861,551): text "SHIFTS"; opens SHIFT
rounded rectangle at (360,470)-(581,551): text "MILLS"; opens MILL
rounded rectangle at (930,470)-(1181,551): text "PROGRAM SETTINGS"; opens PROGRAM_SETTINGS
2 more shapes without text or variables
4 elements of other kinds (tables, trends, ...) not read
*)

(* Visualisation MILL
